(* IEC 61131-3 sources: TIA2AX/tests/V18/test_projects/expected/HW_2200330/ST40_PLC, 7 files *)

(* ---- HwIdentifiers.st ---- *)
TYPE
	HwIdentifiers : WORD
	(
		ST40_PLC_Profilschiene_0 :=	WORD#256,
		ST40_PLC :=	WORD#48,
		ST40_PLC_Card_reader_writer_1 :=	WORD#51,
		ST40_PLC_CPU_display_1 :=	WORD#54,
		ST40_PLC_OPC_UA_1 :=	WORD#117,
		ST40_PLC_DP_interface_1 :=	WORD#60,
		ST40_PLC_PROFINET_interface_1 :=	WORD#64,
		ST40_PLC_PROFINET_interface_1_Port_1 :=	WORD#65,
		ST40_PLC_PROFINET_interface_1_Port_2 :=	WORD#66,
		ST40_PLC_PROFINET_interface_2 :=	WORD#72,
		ST40_PLC_PROFINET_interface_2_Port_1 :=	WORD#73,
		ST40_Switch_SCALANCE_X_rack :=	WORD#415,
		ST40_Switch :=	WORD#416,
		ST40_Switch_ST40_Switch :=	WORD#417,
		ST40_Switch_SCALANCE_interface_1 :=	WORD#418,
		ST40_Switch_SCALANCE_interface_1_Port_1 :=	WORD#419,
		ST40_Switch_SCALANCE_interface_1_Port_2 :=	WORD#420,
		ST40_Switch_SCALANCE_interface_1_Port_3 :=	WORD#421,
		ST40_Switch_SCALANCE_interface_1_Port_4 :=	WORD#422,
		ST40_Switch_SCALANCE_interface_1_Port_5 :=	WORD#423,
		ST40_Switch_SCALANCE_interface_1_Port_6 :=	WORD#424,
		ST40_Switch_SCALANCE_interface_1_Port_7 :=	WORD#425,
		ST40_Switch_SCALANCE_interface_1_Port_8 :=	WORD#426,
		ST40_Switch_SCALANCE_interface_1_Port_9 :=	WORD#427,
		ST40_Switch_SCALANCE_interface_1_Port_10 :=	WORD#428,
		ST40_Switch_SCALANCE_interface_1_Port_11 :=	WORD#429,
		ST40_Switch_SCALANCE_interface_1_Port_12 :=	WORD#430,
		ST40_Switch_SCALANCE_interface_1_Port_13 :=	WORD#431,
		ST40_Switch_SCALANCE_interface_1_Port_14 :=	WORD#432,
		ST40_Switch_SCALANCE_interface_1_Port_15 :=	WORD#433,
		ST40_Switch_SCALANCE_interface_1_Port_16 :=	WORD#434,
		ST40_2_DM260_Rack :=	WORD#270,
		ST40_2_DM260 :=	WORD#258,
		ST40_2_DM260_Interface :=	WORD#259,
		ST40_2_DM260_Interface_Port_1 :=	WORD#260,
		ST40_2_DM260_DataMan_260 :=	WORD#261,
		ST40_2_DM260_Acquisition_Control_1 :=	WORD#262,
		ST40_2_DM260_Acquisition_Status_1 :=	WORD#263,
		ST40_2_DM260_Results_Control_1 :=	WORD#264,
		ST40_2_DM260_Results_Status_1 :=	WORD#265,
		ST40_2_DM260_Soft_Event_Control_1 :=	WORD#266,
		ST40_2_DM260_User_Data_64_bytes_1 :=	WORD#267,
		ST40_2_DM260_Result_Data_64_bytes_1 :=	WORD#268,
		ST40_3_DM260_Rack :=	WORD#272,
		ST40_3_DM260 :=	WORD#273,
		ST40_3_DM260_Interface :=	WORD#274,
		ST40_3_DM260_Interface_Port_1 :=	WORD#275,
		ST40_3_DM260_DataMan_260 :=	WORD#276,
		ST40_3_DM260_Acquisition_Control_1 :=	WORD#277,
		ST40_3_DM260_Acquisition_Status_1 :=	WORD#278,
		ST40_3_DM260_Results_Control_1 :=	WORD#279,
		ST40_3_DM260_Results_Status_1 :=	WORD#280,
		ST40_3_DM260_Soft_Event_Control_1 :=	WORD#281,
		ST40_3_DM260_User_Data_64_bytes_1 :=	WORD#282,
		ST40_3_DM260_Result_Data_64_bytes_1 :=	WORD#283,
		ST40_1_DM260_Rack :=	WORD#285,
		ST40_1_DM260 :=	WORD#286,
		ST40_1_DM260_Interface :=	WORD#287,
		ST40_1_DM260_Interface_Port_1 :=	WORD#288,
		ST40_1_DM260_DataMan_260 :=	WORD#289,
		ST40_1_DM260_Acquisition_Control_1 :=	WORD#290,
		ST40_1_DM260_Acquisition_Status_1 :=	WORD#291,
		ST40_1_DM260_Results_Control_1 :=	WORD#292,
		ST40_1_DM260_Results_Status_1 :=	WORD#293,
		ST40_1_DM260_Soft_Event_Control_1 :=	WORD#294,
		ST40_1_DM260_User_Data_64_bytes_1 :=	WORD#295,
		ST40_1_DM260_Result_Data_64_bytes_1 :=	WORD#296,
		ST40_2_CMMT_2GF2_Promess_PN_IO_Interface :=	WORD#300,
		ST40_2_CMMT_2GF2_Promess_PN_IO_Interface_Port_1 :=	WORD#301,
		ST40_2_CMMT_2GF2_Promess_PN_IO_Interface_Port_2 :=	WORD#302,
		ST40_2_CMMT_2GF2_Promess_CMMT_AS_V1 :=	WORD#303,
		ST40_2_CMMT_2GF2_Promess_DO_SERVO_1_Module_Access_Point :=	WORD#305,
		ST40_2_CMMT_2GF2_Promess_DO_SERVO_1_Siemens_telegram_111_PZD_12_12 :=	WORD#306,
		ST40_2_CMMT_2GF2_Promess_Siemens_telegram_111_PZD_12_12 :=	WORD#306,
		ST40_2_Promess_Rack :=	WORD#328,
		ST40_2_Promess :=	WORD#329,
		ST40_2_Promess_X1 :=	WORD#330,
		ST40_2_Promess_X1_X1_P1 :=	WORD#331,
		ST40_2_Promess_X1_X1_P2 :=	WORD#332,
		ST40_2_Promess_UniDrive_M :=	WORD#333,
		ST40_2_Promess_Menu_30_01_In_1 :=	WORD#334,
		ST40_2_Promess_Menu_30_02_In_1 :=	WORD#335,
		ST40_2_Promess_Menu_30_03_In_1 :=	WORD#336,
		ST40_2_Promess_Menu_30_04_In_1 :=	WORD#337,
		ST40_2_Promess_Menu_30_05_In_1 :=	WORD#338,
		ST40_2_Promess_Menu_30_06_In_1 :=	WORD#339,
		ST40_2_Promess_Menu_30_07_In_1 :=	WORD#340,
		ST40_2_Promess_Menu_30_08_In_1 :=	WORD#341,
		ST40_2_Promess_Menu_30_09_In_1 :=	WORD#342,
		ST40_2_Promess_Menu_30_10_In_1 :=	WORD#343,
		ST40_2_Promess_Menu_30_11_In_1 :=	WORD#344,
		ST40_2_Promess_Menu_30_12_In_1 :=	WORD#345,
		ST40_2_Promess_Menu_30_13_In_1 :=	WORD#346,
		ST40_2_Promess_Menu_30_14_In_1 :=	WORD#347,
		ST40_2_Promess_Menu_30_15_In_1 :=	WORD#348,
		ST40_2_Promess_Menu_30_16_In_1 :=	WORD#349,
		ST40_2_Promess_Menu_30_33_Out_1 :=	WORD#350,
		ST40_2_Promess_Menu_30_34_Out_1 :=	WORD#351,
		ST40_2_Promess_Menu_30_35_Out_1 :=	WORD#352,
		ST40_2_Promess_Menu_30_36_Out_1 :=	WORD#353,
		ST40_2_Promess_Menu_30_37_Out_1 :=	WORD#354,
		ST40_2_Promess_Menu_30_38_Out_1 :=	WORD#355,
		ST40_2_Promess_Menu_30_39_Out_1 :=	WORD#356,
		ST40_2_Promess_Menu_30_40_Out_1 :=	WORD#357,
		ST40_2_Promess_Menu_30_41_Out_1 :=	WORD#358,
		ST40_2_Promess_Menu_30_42_Out_1 :=	WORD#359,
		ST40_2_Promess_Menu_30_43_Out_1 :=	WORD#360,
		ST40_2_Promess_Menu_30_44_Out_1 :=	WORD#361,
		ST40_2_Promess_Menu_30_45_Out_1 :=	WORD#362,
		ST40_2_Promess_Menu_30_46_Out_1 :=	WORD#363,
		ST40_2_Promess_Menu_30_47_Out_1 :=	WORD#364,
		ST40_2_Promess_Menu_30_48_Out_1 :=	WORD#365,
		ST40_2_Promess_Menu_30_17_In_1 :=	WORD#366,
		ST40_2_Promess_Menu_30_18_In_1 :=	WORD#367,
		ST40_2_Promess_Menu_30_19_In_1 :=	WORD#368,
		ST40_2_Promess_Menu_30_20_In_1 :=	WORD#369,
		ST40_2_Promess_Menu_30_21_In_1 :=	WORD#370,
		ST40_2_Promess_Menu_30_22_In_1 :=	WORD#371,
		ST40_2_Promess_Menu_30_23_In_1 :=	WORD#372,
		ST40_2_Promess_Menu_30_24_In_1 :=	WORD#373,
		ST40_2_Promess_Menu_30_25_In_1 :=	WORD#374,
		ST40_2_Promess_Menu_30_26_In_1 :=	WORD#375,
		ST40_2_Promess_Menu_30_27_In_1 :=	WORD#376,
		ST40_2_Promess_Menu_30_28_In_1 :=	WORD#377,
		ST40_2_Promess_Menu_30_29_In_1 :=	WORD#307,
		ST40_2_Promess_Menu_30_30_In_1 :=	WORD#308,
		ST40_2_Promess_Menu_30_31_In_1 :=	WORD#309,
		ST40_2_Promess_Menu_30_32_In_1 :=	WORD#310,
		ST40_2_Promess_Menu_30_49_Out_1 :=	WORD#311,
		ST40_2_Promess_Menu_30_50_Out_1 :=	WORD#312,
		ST40_2_Promess_Menu_30_51_Out_1 :=	WORD#313,
		ST40_2_Promess_Menu_30_52_Out_1 :=	WORD#314,
		ST40_2_Promess_Menu_30_53_Out_1 :=	WORD#315,
		ST40_2_Promess_Menu_30_54_Out_1 :=	WORD#316,
		ST40_2_Promess_Menu_30_55_Out_1 :=	WORD#317,
		ST40_2_Promess_Menu_30_56_Out_1 :=	WORD#318,
		ST40_2_Promess_Menu_30_57_Out_1 :=	WORD#319,
		ST40_2_Promess_Menu_30_58_Out_1 :=	WORD#320,
		ST40_2_Promess_Menu_30_59_Out_1 :=	WORD#321,
		ST40_2_Promess_Menu_30_60_Out_1 :=	WORD#322,
		ST40_2_Promess_Menu_30_61_Out_1 :=	WORD#323,
		ST40_2_Promess_Menu_30_62_Out_1 :=	WORD#324,
		ST40_2_Promess_Menu_30_63_Out_1 :=	WORD#325,
		ST40_2_Promess_Menu_30_64_Out_1 :=	WORD#326,
		ST40_CPX_PN_IO_Interface :=	WORD#381,
		ST40_CPX_PN_IO_Interface_Port_1 :=	WORD#382,
		ST40_CPX_PN_IO_Interface_Port_2 :=	WORD#383,
		ST40_CPX_CPX :=	WORD#384,
		ST40_CPX_MPA1S_VMPA1_FB_EMS_8_8DO_1 :=	WORD#385,
		ST40_CPX_MPA1S_VMPA1_FB_EMS_8_8DO_2 :=	WORD#386,
		ST40_CPX_MPA1S_VMPA1_FB_EMS_8_8DO_3 :=	WORD#387,
		ST40_CPX_MPA1G_VMPA1_FB_EMG_8_8DO_1 :=	WORD#388,
		ST40_ET200SP_Rack_0 :=	WORD#390,
		ST40_ET200SP :=	WORD#391,
		ST40_ET200SP_ST40_ET200SP :=	WORD#392,
		ST40_ET200SP_PROFINET_interface :=	WORD#393,
		ST40_ET200SP_PROFINET_interface_Port_1 :=	WORD#395,
		ST40_ET200SP_PROFINET_interface_Port_2 :=	WORD#394,
		ST40_ET200SP_BA_2xRJ45 :=	WORD#395,
		ST40_ET200SP_CM_4xIO_Link_1 :=	WORD#396,
		ST40_ET200SP_CM_4xIO_Link_2 :=	WORD#397,
		ST40_ET200SP_DI_8x24VDC_ST_1 :=	WORD#398,
		ST40_ET200SP_DI_8x24VDC_ST_2 :=	WORD#399,
		ST40_ET200SP_DI_16x24VDC_ST_1 :=	WORD#400,
		ST40_ET200SP_DI_8x24VDC_ST_3 :=	WORD#401,
		ST40_ET200SP_DQ_16x24VDC_0_5A_ST_1 :=	WORD#402,
		ST40_ET200SP_DQ_8x24VDC_0_5A_ST_2 :=	WORD#403,
		ST40_ET200SP_DQ_8x24VDC_0_5A_ST_3 :=	WORD#404,
		ST40_ET200SP_Servermodul_1 :=	WORD#405,
		ST40_HMI_ConnectionBox_Connection_Box :=	WORD#407,
		ST40_HMI_ConnectionBox :=	WORD#408,
		ST40_HMI_ConnectionBox_ST40_HMI_ConnectionBox :=	WORD#409,
		ST40_HMI_ConnectionBox_SCALANCE_interface_1 :=	WORD#410,
		ST40_HMI_ConnectionBox_SCALANCE_interface_1_Port_1 :=	WORD#411,
		ST40_HMI_ConnectionBox_SCALANCE_interface_1_Port_2 :=	WORD#412,
		ST40_HMI_ConnectionBox_SCALANCE_interface_1_Port_3 :=	WORD#413,
		NONE:= WORD#0
	);
END_TYPE

(* ---- HwInputs.st ---- *)
TYPE
	HwInputs : STRUCT
		ST40_2_DM260_Acquisition_Status_1 AT %B2500 : ARRAY[0..2] OF BYTE;
		ST40_2_DM260_Results_Status_1 AT %B2503 : BYTE;
		ST40_2_DM260_Soft_Event_Control_1 AT %B2504 : BYTE;
		ST40_2_DM260_Result_Data_64_bytes_1 AT %B2510 : ARRAY[0..71] OF BYTE;
		ST40_3_DM260_Acquisition_Status_1 AT %B3500 : ARRAY[0..2] OF BYTE;
		ST40_3_DM260_Results_Status_1 AT %B3503 : BYTE;
		ST40_3_DM260_Soft_Event_Control_1 AT %B3504 : BYTE;
		ST40_3_DM260_Result_Data_64_bytes_1 AT %B3510 : ARRAY[0..71] OF BYTE;
		ST40_1_DM260_Acquisition_Status_1 AT %B1600 : ARRAY[0..2] OF BYTE;
		ST40_1_DM260_Results_Status_1 AT %B1603 : BYTE;
		ST40_1_DM260_Soft_Event_Control_1 AT %B1604 : BYTE;
		ST40_1_DM260_Result_Data_64_bytes_1 AT %B1610 : ARRAY[0..71] OF BYTE;
		ST40_2_CMMT_2GF2_Promess_DO_SERVO_1_Siemens_telegram_111_PZD_12_12 AT %B1100 : ARRAY[0..23] OF BYTE;
		ST40_2_Promess_Menu_30_01_In_1 AT %B2100 : WORD;
		ST40_2_Promess_Menu_30_02_In_1 AT %B2102 : WORD;
		ST40_2_Promess_Menu_30_03_In_1 AT %B2104 : WORD;
		ST40_2_Promess_Menu_30_04_In_1 AT %B2106 : WORD;
		ST40_2_Promess_Menu_30_05_In_1 AT %B2108 : WORD;
		ST40_2_Promess_Menu_30_06_In_1 AT %B2110 : WORD;
		ST40_2_Promess_Menu_30_07_In_1 AT %B2112 : WORD;
		ST40_2_Promess_Menu_30_08_In_1 AT %B2114 : WORD;
		ST40_2_Promess_Menu_30_09_In_1 AT %B2116 : WORD;
		ST40_2_Promess_Menu_30_10_In_1 AT %B2118 : WORD;
		ST40_2_Promess_Menu_30_11_In_1 AT %B2120 : WORD;
		ST40_2_Promess_Menu_30_12_In_1 AT %B2122 : WORD;
		ST40_2_Promess_Menu_30_13_In_1 AT %B2124 : WORD;
		ST40_2_Promess_Menu_30_14_In_1 AT %B2126 : WORD;
		ST40_2_Promess_Menu_30_15_In_1 AT %B2128 : WORD;
		ST40_2_Promess_Menu_30_16_In_1 AT %B2130 : WORD;
		ST40_2_Promess_Menu_30_17_In_1 AT %B2132 : WORD;
		ST40_2_Promess_Menu_30_18_In_1 AT %B2134 : WORD;
		ST40_2_Promess_Menu_30_19_In_1 AT %B2136 : WORD;
		ST40_2_Promess_Menu_30_20_In_1 AT %B2138 : WORD;
		ST40_2_Promess_Menu_30_21_In_1 AT %B2140 : WORD;
		ST40_2_Promess_Menu_30_22_In_1 AT %B2142 : WORD;
		ST40_2_Promess_Menu_30_23_In_1 AT %B2144 : WORD;
		ST40_2_Promess_Menu_30_24_In_1 AT %B2146 : WORD;
		ST40_2_Promess_Menu_30_25_In_1 AT %B2148 : WORD;
		ST40_2_Promess_Menu_30_26_In_1 AT %B2150 : WORD;
		ST40_2_Promess_Menu_30_27_In_1 AT %B2152 : WORD;
		ST40_2_Promess_Menu_30_28_In_1 AT %B2154 : WORD;
		ST40_2_Promess_Menu_30_29_In_1 AT %B2156 : WORD;
		ST40_2_Promess_Menu_30_30_In_1 AT %B2158 : WORD;
		ST40_2_Promess_Menu_30_31_In_1 AT %B2160 : WORD;
		ST40_2_Promess_Menu_30_32_In_1 AT %B2162 : WORD;
		ST40_ET200SP_CM_4xIO_Link_1 AT %B100 : ARRAY[0..31] OF BYTE;
		ST40_ET200SP_CM_4xIO_Link_2 AT %B132 : ARRAY[0..31] OF BYTE;
		ST40_ET200SP_DI_8x24VDC_ST_1 AT %B0 : BYTE;
		ST40_ET200SP_DI_8x24VDC_ST_2 AT %B1 : BYTE;
		ST40_ET200SP_DI_16x24VDC_ST_1 AT %B2 : WORD;
		ST40_ET200SP_DI_8x24VDC_ST_3 AT %B4 : BYTE;
	END_STRUCT;
END_TYPE

(* ---- HwOutputs.st ---- *)
TYPE
	HwOutputs : STRUCT
		ST40_2_DM260_Acquisition_Control_1 AT %B2500 : BYTE;
		ST40_2_DM260_Results_Control_1 AT %B2503 : BYTE;
		ST40_2_DM260_Soft_Event_Control_1 AT %B2504 : BYTE;
		ST40_2_DM260_User_Data_64_bytes_1 AT %B2510 : ARRAY[0..67] OF BYTE;
		ST40_3_DM260_Acquisition_Control_1 AT %B3500 : BYTE;
		ST40_3_DM260_Results_Control_1 AT %B3503 : BYTE;
		ST40_3_DM260_Soft_Event_Control_1 AT %B3504 : BYTE;
		ST40_3_DM260_User_Data_64_bytes_1 AT %B3510 : ARRAY[0..67] OF BYTE;
		ST40_1_DM260_Acquisition_Control_1 AT %B1600 : BYTE;
		ST40_1_DM260_Results_Control_1 AT %B1603 : BYTE;
		ST40_1_DM260_Soft_Event_Control_1 AT %B1604 : BYTE;
		ST40_1_DM260_User_Data_64_bytes_1 AT %B1610 : ARRAY[0..67] OF BYTE;
		ST40_2_CMMT_2GF2_Promess_DO_SERVO_1_Siemens_telegram_111_PZD_12_12 AT %B1100 : ARRAY[0..23] OF BYTE;
		ST40_2_Promess_Menu_30_33_Out_1 AT %B2100 : WORD;
		ST40_2_Promess_Menu_30_34_Out_1 AT %B2102 : WORD;
		ST40_2_Promess_Menu_30_35_Out_1 AT %B2104 : WORD;
		ST40_2_Promess_Menu_30_36_Out_1 AT %B2106 : WORD;
		ST40_2_Promess_Menu_30_37_Out_1 AT %B2108 : WORD;
		ST40_2_Promess_Menu_30_38_Out_1 AT %B2110 : WORD;
		ST40_2_Promess_Menu_30_39_Out_1 AT %B2112 : WORD;
		ST40_2_Promess_Menu_30_40_Out_1 AT %B2114 : WORD;
		ST40_2_Promess_Menu_30_41_Out_1 AT %B2116 : WORD;
		ST40_2_Promess_Menu_30_42_Out_1 AT %B2118 : WORD;
		ST40_2_Promess_Menu_30_43_Out_1 AT %B2120 : WORD;
		ST40_2_Promess_Menu_30_44_Out_1 AT %B2122 : WORD;
		ST40_2_Promess_Menu_30_45_Out_1 AT %B2124 : WORD;
		ST40_2_Promess_Menu_30_46_Out_1 AT %B2126 : WORD;
		ST40_2_Promess_Menu_30_47_Out_1 AT %B2128 : WORD;
		ST40_2_Promess_Menu_30_48_Out_1 AT %B2130 : WORD;
		ST40_2_Promess_Menu_30_49_Out_1 AT %B2132 : WORD;
		ST40_2_Promess_Menu_30_50_Out_1 AT %B2134 : WORD;
		ST40_2_Promess_Menu_30_51_Out_1 AT %B2136 : WORD;
		ST40_2_Promess_Menu_30_52_Out_1 AT %B2138 : WORD;
		ST40_2_Promess_Menu_30_53_Out_1 AT %B2140 : WORD;
		ST40_2_Promess_Menu_30_54_Out_1 AT %B2142 : WORD;
		ST40_2_Promess_Menu_30_55_Out_1 AT %B2144 : WORD;
		ST40_2_Promess_Menu_30_56_Out_1 AT %B2146 : WORD;
		ST40_2_Promess_Menu_30_57_Out_1 AT %B2148 : WORD;
		ST40_2_Promess_Menu_30_58_Out_1 AT %B2150 : WORD;
		ST40_2_Promess_Menu_30_59_Out_1 AT %B2152 : WORD;
		ST40_2_Promess_Menu_30_60_Out_1 AT %B2154 : WORD;
		ST40_2_Promess_Menu_30_61_Out_1 AT %B2156 : WORD;
		ST40_2_Promess_Menu_30_62_Out_1 AT %B2158 : WORD;
		ST40_2_Promess_Menu_30_63_Out_1 AT %B2160 : WORD;
		ST40_2_Promess_Menu_30_64_Out_1 AT %B2162 : WORD;
		ST40_CPX_MPA1S_VMPA1_FB_EMS_8_8DO_1 AT %B200 : BYTE;
		ST40_CPX_MPA1S_VMPA1_FB_EMS_8_8DO_2 AT %B201 : BYTE;
		ST40_CPX_MPA1S_VMPA1_FB_EMS_8_8DO_3 AT %B202 : BYTE;
		ST40_CPX_MPA1G_VMPA1_FB_EMG_8_8DO_1 AT %B203 : BYTE;
		ST40_ET200SP_CM_4xIO_Link_1 AT %B100 : ARRAY[0..31] OF BYTE;
		ST40_ET200SP_CM_4xIO_Link_2 AT %B132 : ARRAY[0..31] OF BYTE;
		ST40_ET200SP_DQ_16x24VDC_0_5A_ST_1 AT %B0 : WORD;
		ST40_ET200SP_DQ_8x24VDC_0_5A_ST_2 AT %B2 : BYTE;
		ST40_ET200SP_DQ_8x24VDC_0_5A_ST_3 AT %B3 : BYTE;
	END_STRUCT;
END_TYPE

(* ---- PlcInputs.st ---- *)
TYPE
	PlcInputs : STRUCT
		ST40_2_DM260_Acquisition_Status_1 : ARRAY[0..2] OF BYTE;
		ST40_2_DM260_Results_Status_1 : BYTE;
		ST40_2_DM260_Soft_Event_Control_1 : BYTE;
		ST40_2_DM260_Result_Data_64_bytes_1 : ARRAY[0..71] OF BYTE;
		ST40_3_DM260_Acquisition_Status_1 : ARRAY[0..2] OF BYTE;
		ST40_3_DM260_Results_Status_1 : BYTE;
		ST40_3_DM260_Soft_Event_Control_1 : BYTE;
		ST40_3_DM260_Result_Data_64_bytes_1 : ARRAY[0..71] OF BYTE;
		ST40_1_DM260_Acquisition_Status_1 : ARRAY[0..2] OF BYTE;
		ST40_1_DM260_Results_Status_1 : BYTE;
		ST40_1_DM260_Soft_Event_Control_1 : BYTE;
		ST40_1_DM260_Result_Data_64_bytes_1 : ARRAY[0..71] OF BYTE;
		ST40_2_CMMT_2GF2_Promess_DO_SERVO_1_Siemens_telegram_111_PZD_12_12 : ARRAY[0..23] OF BYTE;
		ST40_2_Promess_Menu_30_01_In_1 : WORD;
		ST40_2_Promess_Menu_30_02_In_1 : WORD;
		ST40_2_Promess_Menu_30_03_In_1 : WORD;
		ST40_2_Promess_Menu_30_04_In_1 : WORD;
		ST40_2_Promess_Menu_30_05_In_1 : WORD;
		ST40_2_Promess_Menu_30_06_In_1 : WORD;
		ST40_2_Promess_Menu_30_07_In_1 : WORD;
		ST40_2_Promess_Menu_30_08_In_1 : WORD;
		ST40_2_Promess_Menu_30_09_In_1 : WORD;
		ST40_2_Promess_Menu_30_10_In_1 : WORD;
		ST40_2_Promess_Menu_30_11_In_1 : WORD;
		ST40_2_Promess_Menu_30_12_In_1 : WORD;
		ST40_2_Promess_Menu_30_13_In_1 : WORD;
		ST40_2_Promess_Menu_30_14_In_1 : WORD;
		ST40_2_Promess_Menu_30_15_In_1 : WORD;
		ST40_2_Promess_Menu_30_16_In_1 : WORD;
		ST40_2_Promess_Menu_30_17_In_1 : WORD;
		ST40_2_Promess_Menu_30_18_In_1 : WORD;
		ST40_2_Promess_Menu_30_19_In_1 : WORD;
		ST40_2_Promess_Menu_30_20_In_1 : WORD;
		ST40_2_Promess_Menu_30_21_In_1 : WORD;
		ST40_2_Promess_Menu_30_22_In_1 : WORD;
		ST40_2_Promess_Menu_30_23_In_1 : WORD;
		ST40_2_Promess_Menu_30_24_In_1 : WORD;
		ST40_2_Promess_Menu_30_25_In_1 : WORD;
		ST40_2_Promess_Menu_30_26_In_1 : WORD;
		ST40_2_Promess_Menu_30_27_In_1 : WORD;
		ST40_2_Promess_Menu_30_28_In_1 : WORD;
		ST40_2_Promess_Menu_30_29_In_1 : WORD;
		ST40_2_Promess_Menu_30_30_In_1 : WORD;
		ST40_2_Promess_Menu_30_31_In_1 : WORD;
		ST40_2_Promess_Menu_30_32_In_1 : WORD;
		ST40_ET200SP_CM_4xIO_Link_1 : ARRAY[0..31] OF BYTE;
		ST40_ET200SP_CM_4xIO_Link_2 : ARRAY[0..31] OF BYTE;
		ST40_ET200SP_DI_8x24VDC_ST_1 : BYTE;
		ST40_ET200SP_DI_8x24VDC_ST_2 : BYTE;
		ST40_ET200SP_DI_16x24VDC_ST_1 : WORD;
		ST40_ET200SP_DI_8x24VDC_ST_3 : BYTE;
	END_STRUCT;
END_TYPE

(* ---- PlcOutputs.st ---- *)
TYPE
	PlcOutputs : STRUCT
		ST40_2_DM260_Acquisition_Control_1 : BYTE;
		ST40_2_DM260_Results_Control_1 : BYTE;
		ST40_2_DM260_Soft_Event_Control_1 : BYTE;
		ST40_2_DM260_User_Data_64_bytes_1 : ARRAY[0..67] OF BYTE;
		ST40_3_DM260_Acquisition_Control_1 : BYTE;
		ST40_3_DM260_Results_Control_1 : BYTE;
		ST40_3_DM260_Soft_Event_Control_1 : BYTE;
		ST40_3_DM260_User_Data_64_bytes_1 : ARRAY[0..67] OF BYTE;
		ST40_1_DM260_Acquisition_Control_1 : BYTE;
		ST40_1_DM260_Results_Control_1 : BYTE;
		ST40_1_DM260_Soft_Event_Control_1 : BYTE;
		ST40_1_DM260_User_Data_64_bytes_1 : ARRAY[0..67] OF BYTE;
		ST40_2_CMMT_2GF2_Promess_DO_SERVO_1_Siemens_telegram_111_PZD_12_12 : ARRAY[0..23] OF BYTE;
		ST40_2_Promess_Menu_30_33_Out_1 : WORD;
		ST40_2_Promess_Menu_30_34_Out_1 : WORD;
		ST40_2_Promess_Menu_30_35_Out_1 : WORD;
		ST40_2_Promess_Menu_30_36_Out_1 : WORD;
		ST40_2_Promess_Menu_30_37_Out_1 : WORD;
		ST40_2_Promess_Menu_30_38_Out_1 : WORD;
		ST40_2_Promess_Menu_30_39_Out_1 : WORD;
		ST40_2_Promess_Menu_30_40_Out_1 : WORD;
		ST40_2_Promess_Menu_30_41_Out_1 : WORD;
		ST40_2_Promess_Menu_30_42_Out_1 : WORD;
		ST40_2_Promess_Menu_30_43_Out_1 : WORD;
		ST40_2_Promess_Menu_30_44_Out_1 : WORD;
		ST40_2_Promess_Menu_30_45_Out_1 : WORD;
		ST40_2_Promess_Menu_30_46_Out_1 : WORD;
		ST40_2_Promess_Menu_30_47_Out_1 : WORD;
		ST40_2_Promess_Menu_30_48_Out_1 : WORD;
		ST40_2_Promess_Menu_30_49_Out_1 : WORD;
		ST40_2_Promess_Menu_30_50_Out_1 : WORD;
		ST40_2_Promess_Menu_30_51_Out_1 : WORD;
		ST40_2_Promess_Menu_30_52_Out_1 : WORD;
		ST40_2_Promess_Menu_30_53_Out_1 : WORD;
		ST40_2_Promess_Menu_30_54_Out_1 : WORD;
		ST40_2_Promess_Menu_30_55_Out_1 : WORD;
		ST40_2_Promess_Menu_30_56_Out_1 : WORD;
		ST40_2_Promess_Menu_30_57_Out_1 : WORD;
		ST40_2_Promess_Menu_30_58_Out_1 : WORD;
		ST40_2_Promess_Menu_30_59_Out_1 : WORD;
		ST40_2_Promess_Menu_30_60_Out_1 : WORD;
		ST40_2_Promess_Menu_30_61_Out_1 : WORD;
		ST40_2_Promess_Menu_30_62_Out_1 : WORD;
		ST40_2_Promess_Menu_30_63_Out_1 : WORD;
		ST40_2_Promess_Menu_30_64_Out_1 : WORD;
		ST40_CPX_MPA1S_VMPA1_FB_EMS_8_8DO_1 : BYTE;
		ST40_CPX_MPA1S_VMPA1_FB_EMS_8_8DO_2 : BYTE;
		ST40_CPX_MPA1S_VMPA1_FB_EMS_8_8DO_3 : BYTE;
		ST40_CPX_MPA1G_VMPA1_FB_EMG_8_8DO_1 : BYTE;
		ST40_ET200SP_CM_4xIO_Link_1 : ARRAY[0..31] OF BYTE;
		ST40_ET200SP_CM_4xIO_Link_2 : ARRAY[0..31] OF BYTE;
		ST40_ET200SP_DQ_16x24VDC_0_5A_ST_1 : WORD;
		ST40_ET200SP_DQ_8x24VDC_0_5A_ST_2 : BYTE;
		ST40_ET200SP_DQ_8x24VDC_0_5A_ST_3 : BYTE;
	END_STRUCT;
END_TYPE

(* ---- CopyInputs.st ---- *)
FUNCTION CopyInputs
	VAR_EXTERNAL
		HwInputs : HwInputs;
		PlcInputs : PlcInputs;
	END_VAR
	PlcInputs.ST40_2_DM260_Acquisition_Status_1[0] := HwInputs.ST40_2_DM260_Acquisition_Status_1[0];
	PlcInputs.ST40_2_DM260_Acquisition_Status_1[1] := HwInputs.ST40_2_DM260_Acquisition_Status_1[1];
	PlcInputs.ST40_2_DM260_Acquisition_Status_1[2] := HwInputs.ST40_2_DM260_Acquisition_Status_1[2];
	PlcInputs.ST40_2_DM260_Results_Status_1 := HwInputs.ST40_2_DM260_Results_Status_1;
	PlcInputs.ST40_2_DM260_Soft_Event_Control_1 := HwInputs.ST40_2_DM260_Soft_Event_Control_1;
	PlcInputs.ST40_2_DM260_Result_Data_64_bytes_1[0] := HwInputs.ST40_2_DM260_Result_Data_64_bytes_1[0];
	PlcInputs.ST40_2_DM260_Result_Data_64_bytes_1[1] := HwInputs.ST40_2_DM260_Result_Data_64_bytes_1[1];
	PlcInputs.ST40_2_DM260_Result_Data_64_bytes_1[2] := HwInputs.ST40_2_DM260_Result_Data_64_bytes_1[2];
	PlcInputs.ST40_2_DM260_Result_Data_64_bytes_1[3] := HwInputs.ST40_2_DM260_Result_Data_64_bytes_1[3];
	PlcInputs.ST40_2_DM260_Result_Data_64_bytes_1[4] := HwInputs.ST40_2_DM260_Result_Data_64_bytes_1[4];
	PlcInputs.ST40_2_DM260_Result_Data_64_bytes_1[5] := HwInputs.ST40_2_DM260_Result_Data_64_bytes_1[5];
	PlcInputs.ST40_2_DM260_Result_Data_64_bytes_1[6] := HwInputs.ST40_2_DM260_Result_Data_64_bytes_1[6];
	PlcInputs.ST40_2_DM260_Result_Data_64_bytes_1[7] := HwInputs.ST40_2_DM260_Result_Data_64_bytes_1[7];
	PlcInputs.ST40_2_DM260_Result_Data_64_bytes_1[8] := HwInputs.ST40_2_DM260_Result_Data_64_bytes_1[8];
	PlcInputs.ST40_2_DM260_Result_Data_64_bytes_1[9] := HwInputs.ST40_2_DM260_Result_Data_64_bytes_1[9];
	PlcInputs.ST40_2_DM260_Result_Data_64_bytes_1[10] := HwInputs.ST40_2_DM260_Result_Data_64_bytes_1[10];
	PlcInputs.ST40_2_DM260_Result_Data_64_bytes_1[11] := HwInputs.ST40_2_DM260_Result_Data_64_bytes_1[11];
	PlcInputs.ST40_2_DM260_Result_Data_64_bytes_1[12] := HwInputs.ST40_2_DM260_Result_Data_64_bytes_1[12];
	PlcInputs.ST40_2_DM260_Result_Data_64_bytes_1[13] := HwInputs.ST40_2_DM260_Result_Data_64_bytes_1[13];
	PlcInputs.ST40_2_DM260_Result_Data_64_bytes_1[14] := HwInputs.ST40_2_DM260_Result_Data_64_bytes_1[14];
	PlcInputs.ST40_2_DM260_Result_Data_64_bytes_1[15] := HwInputs.ST40_2_DM260_Result_Data_64_bytes_1[15];
	PlcInputs.ST40_2_DM260_Result_Data_64_bytes_1[16] := HwInputs.ST40_2_DM260_Result_Data_64_bytes_1[16];
	PlcInputs.ST40_2_DM260_Result_Data_64_bytes_1[17] := HwInputs.ST40_2_DM260_Result_Data_64_bytes_1[17];
	PlcInputs.ST40_2_DM260_Result_Data_64_bytes_1[18] := HwInputs.ST40_2_DM260_Result_Data_64_bytes_1[18];
	PlcInputs.ST40_2_DM260_Result_Data_64_bytes_1[19] := HwInputs.ST40_2_DM260_Result_Data_64_bytes_1[19];
	PlcInputs.ST40_2_DM260_Result_Data_64_bytes_1[20] := HwInputs.ST40_2_DM260_Result_Data_64_bytes_1[20];
	PlcInputs.ST40_2_DM260_Result_Data_64_bytes_1[21] := HwInputs.ST40_2_DM260_Result_Data_64_bytes_1[21];
	PlcInputs.ST40_2_DM260_Result_Data_64_bytes_1[22] := HwInputs.ST40_2_DM260_Result_Data_64_bytes_1[22];
	PlcInputs.ST40_2_DM260_Result_Data_64_bytes_1[23] := HwInputs.ST40_2_DM260_Result_Data_64_bytes_1[23];
	PlcInputs.ST40_2_DM260_Result_Data_64_bytes_1[24] := HwInputs.ST40_2_DM260_Result_Data_64_bytes_1[24];
	PlcInputs.ST40_2_DM260_Result_Data_64_bytes_1[25] := HwInputs.ST40_2_DM260_Result_Data_64_bytes_1[25];
	PlcInputs.ST40_2_DM260_Result_Data_64_bytes_1[26] := HwInputs.ST40_2_DM260_Result_Data_64_bytes_1[26];
	PlcInputs.ST40_2_DM260_Result_Data_64_bytes_1[27] := HwInputs.ST40_2_DM260_Result_Data_64_bytes_1[27];
	PlcInputs.ST40_2_DM260_Result_Data_64_bytes_1[28] := HwInputs.ST40_2_DM260_Result_Data_64_bytes_1[28];
	PlcInputs.ST40_2_DM260_Result_Data_64_bytes_1[29] := HwInputs.ST40_2_DM260_Result_Data_64_bytes_1[29];
	PlcInputs.ST40_2_DM260_Result_Data_64_bytes_1[30] := HwInputs.ST40_2_DM260_Result_Data_64_bytes_1[30];
	PlcInputs.ST40_2_DM260_Result_Data_64_bytes_1[31] := HwInputs.ST40_2_DM260_Result_Data_64_bytes_1[31];
	PlcInputs.ST40_2_DM260_Result_Data_64_bytes_1[32] := HwInputs.ST40_2_DM260_Result_Data_64_bytes_1[32];
	PlcInputs.ST40_2_DM260_Result_Data_64_bytes_1[33] := HwInputs.ST40_2_DM260_Result_Data_64_bytes_1[33];
	PlcInputs.ST40_2_DM260_Result_Data_64_bytes_1[34] := HwInputs.ST40_2_DM260_Result_Data_64_bytes_1[34];
	PlcInputs.ST40_2_DM260_Result_Data_64_bytes_1[35] := HwInputs.ST40_2_DM260_Result_Data_64_bytes_1[35];
	PlcInputs.ST40_2_DM260_Result_Data_64_bytes_1[36] := HwInputs.ST40_2_DM260_Result_Data_64_bytes_1[36];
	PlcInputs.ST40_2_DM260_Result_Data_64_bytes_1[37] := HwInputs.ST40_2_DM260_Result_Data_64_bytes_1[37];
	PlcInputs.ST40_2_DM260_Result_Data_64_bytes_1[38] := HwInputs.ST40_2_DM260_Result_Data_64_bytes_1[38];
	PlcInputs.ST40_2_DM260_Result_Data_64_bytes_1[39] := HwInputs.ST40_2_DM260_Result_Data_64_bytes_1[39];
	PlcInputs.ST40_2_DM260_Result_Data_64_bytes_1[40] := HwInputs.ST40_2_DM260_Result_Data_64_bytes_1[40];
	PlcInputs.ST40_2_DM260_Result_Data_64_bytes_1[41] := HwInputs.ST40_2_DM260_Result_Data_64_bytes_1[41];
	PlcInputs.ST40_2_DM260_Result_Data_64_bytes_1[42] := HwInputs.ST40_2_DM260_Result_Data_64_bytes_1[42];
	PlcInputs.ST40_2_DM260_Result_Data_64_bytes_1[43] := HwInputs.ST40_2_DM260_Result_Data_64_bytes_1[43];
	PlcInputs.ST40_2_DM260_Result_Data_64_bytes_1[44] := HwInputs.ST40_2_DM260_Result_Data_64_bytes_1[44];
	PlcInputs.ST40_2_DM260_Result_Data_64_bytes_1[45] := HwInputs.ST40_2_DM260_Result_Data_64_bytes_1[45];
	PlcInputs.ST40_2_DM260_Result_Data_64_bytes_1[46] := HwInputs.ST40_2_DM260_Result_Data_64_bytes_1[46];
	PlcInputs.ST40_2_DM260_Result_Data_64_bytes_1[47] := HwInputs.ST40_2_DM260_Result_Data_64_bytes_1[47];
	PlcInputs.ST40_2_DM260_Result_Data_64_bytes_1[48] := HwInputs.ST40_2_DM260_Result_Data_64_bytes_1[48];
	PlcInputs.ST40_2_DM260_Result_Data_64_bytes_1[49] := HwInputs.ST40_2_DM260_Result_Data_64_bytes_1[49];
	PlcInputs.ST40_2_DM260_Result_Data_64_bytes_1[50] := HwInputs.ST40_2_DM260_Result_Data_64_bytes_1[50];
	PlcInputs.ST40_2_DM260_Result_Data_64_bytes_1[51] := HwInputs.ST40_2_DM260_Result_Data_64_bytes_1[51];
	PlcInputs.ST40_2_DM260_Result_Data_64_bytes_1[52] := HwInputs.ST40_2_DM260_Result_Data_64_bytes_1[52];
	PlcInputs.ST40_2_DM260_Result_Data_64_bytes_1[53] := HwInputs.ST40_2_DM260_Result_Data_64_bytes_1[53];
	PlcInputs.ST40_2_DM260_Result_Data_64_bytes_1[54] := HwInputs.ST40_2_DM260_Result_Data_64_bytes_1[54];
	PlcInputs.ST40_2_DM260_Result_Data_64_bytes_1[55] := HwInputs.ST40_2_DM260_Result_Data_64_bytes_1[55];
	PlcInputs.ST40_2_DM260_Result_Data_64_bytes_1[56] := HwInputs.ST40_2_DM260_Result_Data_64_bytes_1[56];
	PlcInputs.ST40_2_DM260_Result_Data_64_bytes_1[57] := HwInputs.ST40_2_DM260_Result_Data_64_bytes_1[57];
	PlcInputs.ST40_2_DM260_Result_Data_64_bytes_1[58] := HwInputs.ST40_2_DM260_Result_Data_64_bytes_1[58];
	PlcInputs.ST40_2_DM260_Result_Data_64_bytes_1[59] := HwInputs.ST40_2_DM260_Result_Data_64_bytes_1[59];
	PlcInputs.ST40_2_DM260_Result_Data_64_bytes_1[60] := HwInputs.ST40_2_DM260_Result_Data_64_bytes_1[60];
	PlcInputs.ST40_2_DM260_Result_Data_64_bytes_1[61] := HwInputs.ST40_2_DM260_Result_Data_64_bytes_1[61];
	PlcInputs.ST40_2_DM260_Result_Data_64_bytes_1[62] := HwInputs.ST40_2_DM260_Result_Data_64_bytes_1[62];
	PlcInputs.ST40_2_DM260_Result_Data_64_bytes_1[63] := HwInputs.ST40_2_DM260_Result_Data_64_bytes_1[63];
	PlcInputs.ST40_2_DM260_Result_Data_64_bytes_1[64] := HwInputs.ST40_2_DM260_Result_Data_64_bytes_1[64];
	PlcInputs.ST40_2_DM260_Result_Data_64_bytes_1[65] := HwInputs.ST40_2_DM260_Result_Data_64_bytes_1[65];
	PlcInputs.ST40_2_DM260_Result_Data_64_bytes_1[66] := HwInputs.ST40_2_DM260_Result_Data_64_bytes_1[66];
	PlcInputs.ST40_2_DM260_Result_Data_64_bytes_1[67] := HwInputs.ST40_2_DM260_Result_Data_64_bytes_1[67];
	PlcInputs.ST40_2_DM260_Result_Data_64_bytes_1[68] := HwInputs.ST40_2_DM260_Result_Data_64_bytes_1[68];
	PlcInputs.ST40_2_DM260_Result_Data_64_bytes_1[69] := HwInputs.ST40_2_DM260_Result_Data_64_bytes_1[69];
	PlcInputs.ST40_2_DM260_Result_Data_64_bytes_1[70] := HwInputs.ST40_2_DM260_Result_Data_64_bytes_1[70];
	PlcInputs.ST40_2_DM260_Result_Data_64_bytes_1[71] := HwInputs.ST40_2_DM260_Result_Data_64_bytes_1[71];
	PlcInputs.ST40_3_DM260_Acquisition_Status_1[0] := HwInputs.ST40_3_DM260_Acquisition_Status_1[0];
	PlcInputs.ST40_3_DM260_Acquisition_Status_1[1] := HwInputs.ST40_3_DM260_Acquisition_Status_1[1];
	PlcInputs.ST40_3_DM260_Acquisition_Status_1[2] := HwInputs.ST40_3_DM260_Acquisition_Status_1[2];
	PlcInputs.ST40_3_DM260_Results_Status_1 := HwInputs.ST40_3_DM260_Results_Status_1;
	PlcInputs.ST40_3_DM260_Soft_Event_Control_1 := HwInputs.ST40_3_DM260_Soft_Event_Control_1;
	PlcInputs.ST40_3_DM260_Result_Data_64_bytes_1[0] := HwInputs.ST40_3_DM260_Result_Data_64_bytes_1[0];
	PlcInputs.ST40_3_DM260_Result_Data_64_bytes_1[1] := HwInputs.ST40_3_DM260_Result_Data_64_bytes_1[1];
	PlcInputs.ST40_3_DM260_Result_Data_64_bytes_1[2] := HwInputs.ST40_3_DM260_Result_Data_64_bytes_1[2];
	PlcInputs.ST40_3_DM260_Result_Data_64_bytes_1[3] := HwInputs.ST40_3_DM260_Result_Data_64_bytes_1[3];
	PlcInputs.ST40_3_DM260_Result_Data_64_bytes_1[4] := HwInputs.ST40_3_DM260_Result_Data_64_bytes_1[4];
	PlcInputs.ST40_3_DM260_Result_Data_64_bytes_1[5] := HwInputs.ST40_3_DM260_Result_Data_64_bytes_1[5];
	PlcInputs.ST40_3_DM260_Result_Data_64_bytes_1[6] := HwInputs.ST40_3_DM260_Result_Data_64_bytes_1[6];
	PlcInputs.ST40_3_DM260_Result_Data_64_bytes_1[7] := HwInputs.ST40_3_DM260_Result_Data_64_bytes_1[7];
	PlcInputs.ST40_3_DM260_Result_Data_64_bytes_1[8] := HwInputs.ST40_3_DM260_Result_Data_64_bytes_1[8];
	PlcInputs.ST40_3_DM260_Result_Data_64_bytes_1[9] := HwInputs.ST40_3_DM260_Result_Data_64_bytes_1[9];
	PlcInputs.ST40_3_DM260_Result_Data_64_bytes_1[10] := HwInputs.ST40_3_DM260_Result_Data_64_bytes_1[10];
	PlcInputs.ST40_3_DM260_Result_Data_64_bytes_1[11] := HwInputs.ST40_3_DM260_Result_Data_64_bytes_1[11];
	PlcInputs.ST40_3_DM260_Result_Data_64_bytes_1[12] := HwInputs.ST40_3_DM260_Result_Data_64_bytes_1[12];
	PlcInputs.ST40_3_DM260_Result_Data_64_bytes_1[13] := HwInputs.ST40_3_DM260_Result_Data_64_bytes_1[13];
	PlcInputs.ST40_3_DM260_Result_Data_64_bytes_1[14] := HwInputs.ST40_3_DM260_Result_Data_64_bytes_1[14];
	PlcInputs.ST40_3_DM260_Result_Data_64_bytes_1[15] := HwInputs.ST40_3_DM260_Result_Data_64_bytes_1[15];
	PlcInputs.ST40_3_DM260_Result_Data_64_bytes_1[16] := HwInputs.ST40_3_DM260_Result_Data_64_bytes_1[16];
	PlcInputs.ST40_3_DM260_Result_Data_64_bytes_1[17] := HwInputs.ST40_3_DM260_Result_Data_64_bytes_1[17];
	PlcInputs.ST40_3_DM260_Result_Data_64_bytes_1[18] := HwInputs.ST40_3_DM260_Result_Data_64_bytes_1[18];
	PlcInputs.ST40_3_DM260_Result_Data_64_bytes_1[19] := HwInputs.ST40_3_DM260_Result_Data_64_bytes_1[19];
	PlcInputs.ST40_3_DM260_Result_Data_64_bytes_1[20] := HwInputs.ST40_3_DM260_Result_Data_64_bytes_1[20];
	PlcInputs.ST40_3_DM260_Result_Data_64_bytes_1[21] := HwInputs.ST40_3_DM260_Result_Data_64_bytes_1[21];
	PlcInputs.ST40_3_DM260_Result_Data_64_bytes_1[22] := HwInputs.ST40_3_DM260_Result_Data_64_bytes_1[22];
	PlcInputs.ST40_3_DM260_Result_Data_64_bytes_1[23] := HwInputs.ST40_3_DM260_Result_Data_64_bytes_1[23];
	PlcInputs.ST40_3_DM260_Result_Data_64_bytes_1[24] := HwInputs.ST40_3_DM260_Result_Data_64_bytes_1[24];
	PlcInputs.ST40_3_DM260_Result_Data_64_bytes_1[25] := HwInputs.ST40_3_DM260_Result_Data_64_bytes_1[25];
	PlcInputs.ST40_3_DM260_Result_Data_64_bytes_1[26] := HwInputs.ST40_3_DM260_Result_Data_64_bytes_1[26];
	PlcInputs.ST40_3_DM260_Result_Data_64_bytes_1[27] := HwInputs.ST40_3_DM260_Result_Data_64_bytes_1[27];
	PlcInputs.ST40_3_DM260_Result_Data_64_bytes_1[28] := HwInputs.ST40_3_DM260_Result_Data_64_bytes_1[28];
	PlcInputs.ST40_3_DM260_Result_Data_64_bytes_1[29] := HwInputs.ST40_3_DM260_Result_Data_64_bytes_1[29];
	PlcInputs.ST40_3_DM260_Result_Data_64_bytes_1[30] := HwInputs.ST40_3_DM260_Result_Data_64_bytes_1[30];
	PlcInputs.ST40_3_DM260_Result_Data_64_bytes_1[31] := HwInputs.ST40_3_DM260_Result_Data_64_bytes_1[31];
	PlcInputs.ST40_3_DM260_Result_Data_64_bytes_1[32] := HwInputs.ST40_3_DM260_Result_Data_64_bytes_1[32];
	PlcInputs.ST40_3_DM260_Result_Data_64_bytes_1[33] := HwInputs.ST40_3_DM260_Result_Data_64_bytes_1[33];
	PlcInputs.ST40_3_DM260_Result_Data_64_bytes_1[34] := HwInputs.ST40_3_DM260_Result_Data_64_bytes_1[34];
	PlcInputs.ST40_3_DM260_Result_Data_64_bytes_1[35] := HwInputs.ST40_3_DM260_Result_Data_64_bytes_1[35];
	PlcInputs.ST40_3_DM260_Result_Data_64_bytes_1[36] := HwInputs.ST40_3_DM260_Result_Data_64_bytes_1[36];
	PlcInputs.ST40_3_DM260_Result_Data_64_bytes_1[37] := HwInputs.ST40_3_DM260_Result_Data_64_bytes_1[37];
	PlcInputs.ST40_3_DM260_Result_Data_64_bytes_1[38] := HwInputs.ST40_3_DM260_Result_Data_64_bytes_1[38];
	PlcInputs.ST40_3_DM260_Result_Data_64_bytes_1[39] := HwInputs.ST40_3_DM260_Result_Data_64_bytes_1[39];
	PlcInputs.ST40_3_DM260_Result_Data_64_bytes_1[40] := HwInputs.ST40_3_DM260_Result_Data_64_bytes_1[40];
	PlcInputs.ST40_3_DM260_Result_Data_64_bytes_1[41] := HwInputs.ST40_3_DM260_Result_Data_64_bytes_1[41];
	PlcInputs.ST40_3_DM260_Result_Data_64_bytes_1[42] := HwInputs.ST40_3_DM260_Result_Data_64_bytes_1[42];
	PlcInputs.ST40_3_DM260_Result_Data_64_bytes_1[43] := HwInputs.ST40_3_DM260_Result_Data_64_bytes_1[43];
	PlcInputs.ST40_3_DM260_Result_Data_64_bytes_1[44] := HwInputs.ST40_3_DM260_Result_Data_64_bytes_1[44];
	PlcInputs.ST40_3_DM260_Result_Data_64_bytes_1[45] := HwInputs.ST40_3_DM260_Result_Data_64_bytes_1[45];
	PlcInputs.ST40_3_DM260_Result_Data_64_bytes_1[46] := HwInputs.ST40_3_DM260_Result_Data_64_bytes_1[46];
	PlcInputs.ST40_3_DM260_Result_Data_64_bytes_1[47] := HwInputs.ST40_3_DM260_Result_Data_64_bytes_1[47];
	PlcInputs.ST40_3_DM260_Result_Data_64_bytes_1[48] := HwInputs.ST40_3_DM260_Result_Data_64_bytes_1[48];
	PlcInputs.ST40_3_DM260_Result_Data_64_bytes_1[49] := HwInputs.ST40_3_DM260_Result_Data_64_bytes_1[49];
	PlcInputs.ST40_3_DM260_Result_Data_64_bytes_1[50] := HwInputs.ST40_3_DM260_Result_Data_64_bytes_1[50];
	PlcInputs.ST40_3_DM260_Result_Data_64_bytes_1[51] := HwInputs.ST40_3_DM260_Result_Data_64_bytes_1[51];
	PlcInputs.ST40_3_DM260_Result_Data_64_bytes_1[52] := HwInputs.ST40_3_DM260_Result_Data_64_bytes_1[52];
	PlcInputs.ST40_3_DM260_Result_Data_64_bytes_1[53] := HwInputs.ST40_3_DM260_Result_Data_64_bytes_1[53];
	PlcInputs.ST40_3_DM260_Result_Data_64_bytes_1[54] := HwInputs.ST40_3_DM260_Result_Data_64_bytes_1[54];
	PlcInputs.ST40_3_DM260_Result_Data_64_bytes_1[55] := HwInputs.ST40_3_DM260_Result_Data_64_bytes_1[55];
	PlcInputs.ST40_3_DM260_Result_Data_64_bytes_1[56] := HwInputs.ST40_3_DM260_Result_Data_64_bytes_1[56];
	PlcInputs.ST40_3_DM260_Result_Data_64_bytes_1[57] := HwInputs.ST40_3_DM260_Result_Data_64_bytes_1[57];
	PlcInputs.ST40_3_DM260_Result_Data_64_bytes_1[58] := HwInputs.ST40_3_DM260_Result_Data_64_bytes_1[58];
	PlcInputs.ST40_3_DM260_Result_Data_64_bytes_1[59] := HwInputs.ST40_3_DM260_Result_Data_64_bytes_1[59];
	PlcInputs.ST40_3_DM260_Result_Data_64_bytes_1[60] := HwInputs.ST40_3_DM260_Result_Data_64_bytes_1[60];
	PlcInputs.ST40_3_DM260_Result_Data_64_bytes_1[61] := HwInputs.ST40_3_DM260_Result_Data_64_bytes_1[61];
	PlcInputs.ST40_3_DM260_Result_Data_64_bytes_1[62] := HwInputs.ST40_3_DM260_Result_Data_64_bytes_1[62];
	PlcInputs.ST40_3_DM260_Result_Data_64_bytes_1[63] := HwInputs.ST40_3_DM260_Result_Data_64_bytes_1[63];
	PlcInputs.ST40_3_DM260_Result_Data_64_bytes_1[64] := HwInputs.ST40_3_DM260_Result_Data_64_bytes_1[64];
	PlcInputs.ST40_3_DM260_Result_Data_64_bytes_1[65] := HwInputs.ST40_3_DM260_Result_Data_64_bytes_1[65];
	PlcInputs.ST40_3_DM260_Result_Data_64_bytes_1[66] := HwInputs.ST40_3_DM260_Result_Data_64_bytes_1[66];
	PlcInputs.ST40_3_DM260_Result_Data_64_bytes_1[67] := HwInputs.ST40_3_DM260_Result_Data_64_bytes_1[67];
	PlcInputs.ST40_3_DM260_Result_Data_64_bytes_1[68] := HwInputs.ST40_3_DM260_Result_Data_64_bytes_1[68];
	PlcInputs.ST40_3_DM260_Result_Data_64_bytes_1[69] := HwInputs.ST40_3_DM260_Result_Data_64_bytes_1[69];
	PlcInputs.ST40_3_DM260_Result_Data_64_bytes_1[70] := HwInputs.ST40_3_DM260_Result_Data_64_bytes_1[70];
	PlcInputs.ST40_3_DM260_Result_Data_64_bytes_1[71] := HwInputs.ST40_3_DM260_Result_Data_64_bytes_1[71];
	PlcInputs.ST40_1_DM260_Acquisition_Status_1[0] := HwInputs.ST40_1_DM260_Acquisition_Status_1[0];
	PlcInputs.ST40_1_DM260_Acquisition_Status_1[1] := HwInputs.ST40_1_DM260_Acquisition_Status_1[1];
	PlcInputs.ST40_1_DM260_Acquisition_Status_1[2] := HwInputs.ST40_1_DM260_Acquisition_Status_1[2];
	PlcInputs.ST40_1_DM260_Results_Status_1 := HwInputs.ST40_1_DM260_Results_Status_1;
	PlcInputs.ST40_1_DM260_Soft_Event_Control_1 := HwInputs.ST40_1_DM260_Soft_Event_Control_1;
	PlcInputs.ST40_1_DM260_Result_Data_64_bytes_1[0] := HwInputs.ST40_1_DM260_Result_Data_64_bytes_1[0];
	PlcInputs.ST40_1_DM260_Result_Data_64_bytes_1[1] := HwInputs.ST40_1_DM260_Result_Data_64_bytes_1[1];
	PlcInputs.ST40_1_DM260_Result_Data_64_bytes_1[2] := HwInputs.ST40_1_DM260_Result_Data_64_bytes_1[2];
	PlcInputs.ST40_1_DM260_Result_Data_64_bytes_1[3] := HwInputs.ST40_1_DM260_Result_Data_64_bytes_1[3];
	PlcInputs.ST40_1_DM260_Result_Data_64_bytes_1[4] := HwInputs.ST40_1_DM260_Result_Data_64_bytes_1[4];
	PlcInputs.ST40_1_DM260_Result_Data_64_bytes_1[5] := HwInputs.ST40_1_DM260_Result_Data_64_bytes_1[5];
	PlcInputs.ST40_1_DM260_Result_Data_64_bytes_1[6] := HwInputs.ST40_1_DM260_Result_Data_64_bytes_1[6];
	PlcInputs.ST40_1_DM260_Result_Data_64_bytes_1[7] := HwInputs.ST40_1_DM260_Result_Data_64_bytes_1[7];
	PlcInputs.ST40_1_DM260_Result_Data_64_bytes_1[8] := HwInputs.ST40_1_DM260_Result_Data_64_bytes_1[8];
	PlcInputs.ST40_1_DM260_Result_Data_64_bytes_1[9] := HwInputs.ST40_1_DM260_Result_Data_64_bytes_1[9];
	PlcInputs.ST40_1_DM260_Result_Data_64_bytes_1[10] := HwInputs.ST40_1_DM260_Result_Data_64_bytes_1[10];
	PlcInputs.ST40_1_DM260_Result_Data_64_bytes_1[11] := HwInputs.ST40_1_DM260_Result_Data_64_bytes_1[11];
	PlcInputs.ST40_1_DM260_Result_Data_64_bytes_1[12] := HwInputs.ST40_1_DM260_Result_Data_64_bytes_1[12];
	PlcInputs.ST40_1_DM260_Result_Data_64_bytes_1[13] := HwInputs.ST40_1_DM260_Result_Data_64_bytes_1[13];
	PlcInputs.ST40_1_DM260_Result_Data_64_bytes_1[14] := HwInputs.ST40_1_DM260_Result_Data_64_bytes_1[14];
	PlcInputs.ST40_1_DM260_Result_Data_64_bytes_1[15] := HwInputs.ST40_1_DM260_Result_Data_64_bytes_1[15];
	PlcInputs.ST40_1_DM260_Result_Data_64_bytes_1[16] := HwInputs.ST40_1_DM260_Result_Data_64_bytes_1[16];
	PlcInputs.ST40_1_DM260_Result_Data_64_bytes_1[17] := HwInputs.ST40_1_DM260_Result_Data_64_bytes_1[17];
	PlcInputs.ST40_1_DM260_Result_Data_64_bytes_1[18] := HwInputs.ST40_1_DM260_Result_Data_64_bytes_1[18];
	PlcInputs.ST40_1_DM260_Result_Data_64_bytes_1[19] := HwInputs.ST40_1_DM260_Result_Data_64_bytes_1[19];
	PlcInputs.ST40_1_DM260_Result_Data_64_bytes_1[20] := HwInputs.ST40_1_DM260_Result_Data_64_bytes_1[20];
	PlcInputs.ST40_1_DM260_Result_Data_64_bytes_1[21] := HwInputs.ST40_1_DM260_Result_Data_64_bytes_1[21];
	PlcInputs.ST40_1_DM260_Result_Data_64_bytes_1[22] := HwInputs.ST40_1_DM260_Result_Data_64_bytes_1[22];
	PlcInputs.ST40_1_DM260_Result_Data_64_bytes_1[23] := HwInputs.ST40_1_DM260_Result_Data_64_bytes_1[23];
	PlcInputs.ST40_1_DM260_Result_Data_64_bytes_1[24] := HwInputs.ST40_1_DM260_Result_Data_64_bytes_1[24];
	PlcInputs.ST40_1_DM260_Result_Data_64_bytes_1[25] := HwInputs.ST40_1_DM260_Result_Data_64_bytes_1[25];
	PlcInputs.ST40_1_DM260_Result_Data_64_bytes_1[26] := HwInputs.ST40_1_DM260_Result_Data_64_bytes_1[26];
	PlcInputs.ST40_1_DM260_Result_Data_64_bytes_1[27] := HwInputs.ST40_1_DM260_Result_Data_64_bytes_1[27];
	PlcInputs.ST40_1_DM260_Result_Data_64_bytes_1[28] := HwInputs.ST40_1_DM260_Result_Data_64_bytes_1[28];
	PlcInputs.ST40_1_DM260_Result_Data_64_bytes_1[29] := HwInputs.ST40_1_DM260_Result_Data_64_bytes_1[29];
	PlcInputs.ST40_1_DM260_Result_Data_64_bytes_1[30] := HwInputs.ST40_1_DM260_Result_Data_64_bytes_1[30];
	PlcInputs.ST40_1_DM260_Result_Data_64_bytes_1[31] := HwInputs.ST40_1_DM260_Result_Data_64_bytes_1[31];
	PlcInputs.ST40_1_DM260_Result_Data_64_bytes_1[32] := HwInputs.ST40_1_DM260_Result_Data_64_bytes_1[32];
	PlcInputs.ST40_1_DM260_Result_Data_64_bytes_1[33] := HwInputs.ST40_1_DM260_Result_Data_64_bytes_1[33];
	PlcInputs.ST40_1_DM260_Result_Data_64_bytes_1[34] := HwInputs.ST40_1_DM260_Result_Data_64_bytes_1[34];
	PlcInputs.ST40_1_DM260_Result_Data_64_bytes_1[35] := HwInputs.ST40_1_DM260_Result_Data_64_bytes_1[35];
	PlcInputs.ST40_1_DM260_Result_Data_64_bytes_1[36] := HwInputs.ST40_1_DM260_Result_Data_64_bytes_1[36];
	PlcInputs.ST40_1_DM260_Result_Data_64_bytes_1[37] := HwInputs.ST40_1_DM260_Result_Data_64_bytes_1[37];
	PlcInputs.ST40_1_DM260_Result_Data_64_bytes_1[38] := HwInputs.ST40_1_DM260_Result_Data_64_bytes_1[38];
	PlcInputs.ST40_1_DM260_Result_Data_64_bytes_1[39] := HwInputs.ST40_1_DM260_Result_Data_64_bytes_1[39];
	PlcInputs.ST40_1_DM260_Result_Data_64_bytes_1[40] := HwInputs.ST40_1_DM260_Result_Data_64_bytes_1[40];
	PlcInputs.ST40_1_DM260_Result_Data_64_bytes_1[41] := HwInputs.ST40_1_DM260_Result_Data_64_bytes_1[41];
	PlcInputs.ST40_1_DM260_Result_Data_64_bytes_1[42] := HwInputs.ST40_1_DM260_Result_Data_64_bytes_1[42];
	PlcInputs.ST40_1_DM260_Result_Data_64_bytes_1[43] := HwInputs.ST40_1_DM260_Result_Data_64_bytes_1[43];
	PlcInputs.ST40_1_DM260_Result_Data_64_bytes_1[44] := HwInputs.ST40_1_DM260_Result_Data_64_bytes_1[44];
	PlcInputs.ST40_1_DM260_Result_Data_64_bytes_1[45] := HwInputs.ST40_1_DM260_Result_Data_64_bytes_1[45];
	PlcInputs.ST40_1_DM260_Result_Data_64_bytes_1[46] := HwInputs.ST40_1_DM260_Result_Data_64_bytes_1[46];
	PlcInputs.ST40_1_DM260_Result_Data_64_bytes_1[47] := HwInputs.ST40_1_DM260_Result_Data_64_bytes_1[47];
	PlcInputs.ST40_1_DM260_Result_Data_64_bytes_1[48] := HwInputs.ST40_1_DM260_Result_Data_64_bytes_1[48];
	PlcInputs.ST40_1_DM260_Result_Data_64_bytes_1[49] := HwInputs.ST40_1_DM260_Result_Data_64_bytes_1[49];
	PlcInputs.ST40_1_DM260_Result_Data_64_bytes_1[50] := HwInputs.ST40_1_DM260_Result_Data_64_bytes_1[50];
	PlcInputs.ST40_1_DM260_Result_Data_64_bytes_1[51] := HwInputs.ST40_1_DM260_Result_Data_64_bytes_1[51];
	PlcInputs.ST40_1_DM260_Result_Data_64_bytes_1[52] := HwInputs.ST40_1_DM260_Result_Data_64_bytes_1[52];
	PlcInputs.ST40_1_DM260_Result_Data_64_bytes_1[53] := HwInputs.ST40_1_DM260_Result_Data_64_bytes_1[53];
	PlcInputs.ST40_1_DM260_Result_Data_64_bytes_1[54] := HwInputs.ST40_1_DM260_Result_Data_64_bytes_1[54];
	PlcInputs.ST40_1_DM260_Result_Data_64_bytes_1[55] := HwInputs.ST40_1_DM260_Result_Data_64_bytes_1[55];
	PlcInputs.ST40_1_DM260_Result_Data_64_bytes_1[56] := HwInputs.ST40_1_DM260_Result_Data_64_bytes_1[56];
	PlcInputs.ST40_1_DM260_Result_Data_64_bytes_1[57] := HwInputs.ST40_1_DM260_Result_Data_64_bytes_1[57];
	PlcInputs.ST40_1_DM260_Result_Data_64_bytes_1[58] := HwInputs.ST40_1_DM260_Result_Data_64_bytes_1[58];
	PlcInputs.ST40_1_DM260_Result_Data_64_bytes_1[59] := HwInputs.ST40_1_DM260_Result_Data_64_bytes_1[59];
	PlcInputs.ST40_1_DM260_Result_Data_64_bytes_1[60] := HwInputs.ST40_1_DM260_Result_Data_64_bytes_1[60];
	PlcInputs.ST40_1_DM260_Result_Data_64_bytes_1[61] := HwInputs.ST40_1_DM260_Result_Data_64_bytes_1[61];
	PlcInputs.ST40_1_DM260_Result_Data_64_bytes_1[62] := HwInputs.ST40_1_DM260_Result_Data_64_bytes_1[62];
	PlcInputs.ST40_1_DM260_Result_Data_64_bytes_1[63] := HwInputs.ST40_1_DM260_Result_Data_64_bytes_1[63];
	PlcInputs.ST40_1_DM260_Result_Data_64_bytes_1[64] := HwInputs.ST40_1_DM260_Result_Data_64_bytes_1[64];
	PlcInputs.ST40_1_DM260_Result_Data_64_bytes_1[65] := HwInputs.ST40_1_DM260_Result_Data_64_bytes_1[65];
	PlcInputs.ST40_1_DM260_Result_Data_64_bytes_1[66] := HwInputs.ST40_1_DM260_Result_Data_64_bytes_1[66];
	PlcInputs.ST40_1_DM260_Result_Data_64_bytes_1[67] := HwInputs.ST40_1_DM260_Result_Data_64_bytes_1[67];
	PlcInputs.ST40_1_DM260_Result_Data_64_bytes_1[68] := HwInputs.ST40_1_DM260_Result_Data_64_bytes_1[68];
	PlcInputs.ST40_1_DM260_Result_Data_64_bytes_1[69] := HwInputs.ST40_1_DM260_Result_Data_64_bytes_1[69];
	PlcInputs.ST40_1_DM260_Result_Data_64_bytes_1[70] := HwInputs.ST40_1_DM260_Result_Data_64_bytes_1[70];
	PlcInputs.ST40_1_DM260_Result_Data_64_bytes_1[71] := HwInputs.ST40_1_DM260_Result_Data_64_bytes_1[71];
	PlcInputs.ST40_2_CMMT_2GF2_Promess_DO_SERVO_1_Siemens_telegram_111_PZD_12_12[0] := HwInputs.ST40_2_CMMT_2GF2_Promess_DO_SERVO_1_Siemens_telegram_111_PZD_12_12[0];
	PlcInputs.ST40_2_CMMT_2GF2_Promess_DO_SERVO_1_Siemens_telegram_111_PZD_12_12[1] := HwInputs.ST40_2_CMMT_2GF2_Promess_DO_SERVO_1_Siemens_telegram_111_PZD_12_12[1];
	PlcInputs.ST40_2_CMMT_2GF2_Promess_DO_SERVO_1_Siemens_telegram_111_PZD_12_12[2] := HwInputs.ST40_2_CMMT_2GF2_Promess_DO_SERVO_1_Siemens_telegram_111_PZD_12_12[2];
	PlcInputs.ST40_2_CMMT_2GF2_Promess_DO_SERVO_1_Siemens_telegram_111_PZD_12_12[3] := HwInputs.ST40_2_CMMT_2GF2_Promess_DO_SERVO_1_Siemens_telegram_111_PZD_12_12[3];
	PlcInputs.ST40_2_CMMT_2GF2_Promess_DO_SERVO_1_Siemens_telegram_111_PZD_12_12[4] := HwInputs.ST40_2_CMMT_2GF2_Promess_DO_SERVO_1_Siemens_telegram_111_PZD_12_12[4];
	PlcInputs.ST40_2_CMMT_2GF2_Promess_DO_SERVO_1_Siemens_telegram_111_PZD_12_12[5] := HwInputs.ST40_2_CMMT_2GF2_Promess_DO_SERVO_1_Siemens_telegram_111_PZD_12_12[5];
	PlcInputs.ST40_2_CMMT_2GF2_Promess_DO_SERVO_1_Siemens_telegram_111_PZD_12_12[6] := HwInputs.ST40_2_CMMT_2GF2_Promess_DO_SERVO_1_Siemens_telegram_111_PZD_12_12[6];
	PlcInputs.ST40_2_CMMT_2GF2_Promess_DO_SERVO_1_Siemens_telegram_111_PZD_12_12[7] := HwInputs.ST40_2_CMMT_2GF2_Promess_DO_SERVO_1_Siemens_telegram_111_PZD_12_12[7];
	PlcInputs.ST40_2_CMMT_2GF2_Promess_DO_SERVO_1_Siemens_telegram_111_PZD_12_12[8] := HwInputs.ST40_2_CMMT_2GF2_Promess_DO_SERVO_1_Siemens_telegram_111_PZD_12_12[8];
	PlcInputs.ST40_2_CMMT_2GF2_Promess_DO_SERVO_1_Siemens_telegram_111_PZD_12_12[9] := HwInputs.ST40_2_CMMT_2GF2_Promess_DO_SERVO_1_Siemens_telegram_111_PZD_12_12[9];
	PlcInputs.ST40_2_CMMT_2GF2_Promess_DO_SERVO_1_Siemens_telegram_111_PZD_12_12[10] := HwInputs.ST40_2_CMMT_2GF2_Promess_DO_SERVO_1_Siemens_telegram_111_PZD_12_12[10];
	PlcInputs.ST40_2_CMMT_2GF2_Promess_DO_SERVO_1_Siemens_telegram_111_PZD_12_12[11] := HwInputs.ST40_2_CMMT_2GF2_Promess_DO_SERVO_1_Siemens_telegram_111_PZD_12_12[11];
	PlcInputs.ST40_2_CMMT_2GF2_Promess_DO_SERVO_1_Siemens_telegram_111_PZD_12_12[12] := HwInputs.ST40_2_CMMT_2GF2_Promess_DO_SERVO_1_Siemens_telegram_111_PZD_12_12[12];
	PlcInputs.ST40_2_CMMT_2GF2_Promess_DO_SERVO_1_Siemens_telegram_111_PZD_12_12[13] := HwInputs.ST40_2_CMMT_2GF2_Promess_DO_SERVO_1_Siemens_telegram_111_PZD_12_12[13];
	PlcInputs.ST40_2_CMMT_2GF2_Promess_DO_SERVO_1_Siemens_telegram_111_PZD_12_12[14] := HwInputs.ST40_2_CMMT_2GF2_Promess_DO_SERVO_1_Siemens_telegram_111_PZD_12_12[14];
	PlcInputs.ST40_2_CMMT_2GF2_Promess_DO_SERVO_1_Siemens_telegram_111_PZD_12_12[15] := HwInputs.ST40_2_CMMT_2GF2_Promess_DO_SERVO_1_Siemens_telegram_111_PZD_12_12[15];
	PlcInputs.ST40_2_CMMT_2GF2_Promess_DO_SERVO_1_Siemens_telegram_111_PZD_12_12[16] := HwInputs.ST40_2_CMMT_2GF2_Promess_DO_SERVO_1_Siemens_telegram_111_PZD_12_12[16];
	PlcInputs.ST40_2_CMMT_2GF2_Promess_DO_SERVO_1_Siemens_telegram_111_PZD_12_12[17] := HwInputs.ST40_2_CMMT_2GF2_Promess_DO_SERVO_1_Siemens_telegram_111_PZD_12_12[17];
	PlcInputs.ST40_2_CMMT_2GF2_Promess_DO_SERVO_1_Siemens_telegram_111_PZD_12_12[18] := HwInputs.ST40_2_CMMT_2GF2_Promess_DO_SERVO_1_Siemens_telegram_111_PZD_12_12[18];
	PlcInputs.ST40_2_CMMT_2GF2_Promess_DO_SERVO_1_Siemens_telegram_111_PZD_12_12[19] := HwInputs.ST40_2_CMMT_2GF2_Promess_DO_SERVO_1_Siemens_telegram_111_PZD_12_12[19];
	PlcInputs.ST40_2_CMMT_2GF2_Promess_DO_SERVO_1_Siemens_telegram_111_PZD_12_12[20] := HwInputs.ST40_2_CMMT_2GF2_Promess_DO_SERVO_1_Siemens_telegram_111_PZD_12_12[20];
	PlcInputs.ST40_2_CMMT_2GF2_Promess_DO_SERVO_1_Siemens_telegram_111_PZD_12_12[21] := HwInputs.ST40_2_CMMT_2GF2_Promess_DO_SERVO_1_Siemens_telegram_111_PZD_12_12[21];
	PlcInputs.ST40_2_CMMT_2GF2_Promess_DO_SERVO_1_Siemens_telegram_111_PZD_12_12[22] := HwInputs.ST40_2_CMMT_2GF2_Promess_DO_SERVO_1_Siemens_telegram_111_PZD_12_12[22];
	PlcInputs.ST40_2_CMMT_2GF2_Promess_DO_SERVO_1_Siemens_telegram_111_PZD_12_12[23] := HwInputs.ST40_2_CMMT_2GF2_Promess_DO_SERVO_1_Siemens_telegram_111_PZD_12_12[23];
	PlcInputs.ST40_2_Promess_Menu_30_01_In_1 := HwInputs.ST40_2_Promess_Menu_30_01_In_1;
	PlcInputs.ST40_2_Promess_Menu_30_02_In_1 := HwInputs.ST40_2_Promess_Menu_30_02_In_1;
	PlcInputs.ST40_2_Promess_Menu_30_03_In_1 := HwInputs.ST40_2_Promess_Menu_30_03_In_1;
	PlcInputs.ST40_2_Promess_Menu_30_04_In_1 := HwInputs.ST40_2_Promess_Menu_30_04_In_1;
	PlcInputs.ST40_2_Promess_Menu_30_05_In_1 := HwInputs.ST40_2_Promess_Menu_30_05_In_1;
	PlcInputs.ST40_2_Promess_Menu_30_06_In_1 := HwInputs.ST40_2_Promess_Menu_30_06_In_1;
	PlcInputs.ST40_2_Promess_Menu_30_07_In_1 := HwInputs.ST40_2_Promess_Menu_30_07_In_1;
	PlcInputs.ST40_2_Promess_Menu_30_08_In_1 := HwInputs.ST40_2_Promess_Menu_30_08_In_1;
	PlcInputs.ST40_2_Promess_Menu_30_09_In_1 := HwInputs.ST40_2_Promess_Menu_30_09_In_1;
	PlcInputs.ST40_2_Promess_Menu_30_10_In_1 := HwInputs.ST40_2_Promess_Menu_30_10_In_1;
	PlcInputs.ST40_2_Promess_Menu_30_11_In_1 := HwInputs.ST40_2_Promess_Menu_30_11_In_1;
	PlcInputs.ST40_2_Promess_Menu_30_12_In_1 := HwInputs.ST40_2_Promess_Menu_30_12_In_1;
	PlcInputs.ST40_2_Promess_Menu_30_13_In_1 := HwInputs.ST40_2_Promess_Menu_30_13_In_1;
	PlcInputs.ST40_2_Promess_Menu_30_14_In_1 := HwInputs.ST40_2_Promess_Menu_30_14_In_1;
	PlcInputs.ST40_2_Promess_Menu_30_15_In_1 := HwInputs.ST40_2_Promess_Menu_30_15_In_1;
	PlcInputs.ST40_2_Promess_Menu_30_16_In_1 := HwInputs.ST40_2_Promess_Menu_30_16_In_1;
	PlcInputs.ST40_2_Promess_Menu_30_17_In_1 := HwInputs.ST40_2_Promess_Menu_30_17_In_1;
	PlcInputs.ST40_2_Promess_Menu_30_18_In_1 := HwInputs.ST40_2_Promess_Menu_30_18_In_1;
	PlcInputs.ST40_2_Promess_Menu_30_19_In_1 := HwInputs.ST40_2_Promess_Menu_30_19_In_1;
	PlcInputs.ST40_2_Promess_Menu_30_20_In_1 := HwInputs.ST40_2_Promess_Menu_30_20_In_1;
	PlcInputs.ST40_2_Promess_Menu_30_21_In_1 := HwInputs.ST40_2_Promess_Menu_30_21_In_1;
	PlcInputs.ST40_2_Promess_Menu_30_22_In_1 := HwInputs.ST40_2_Promess_Menu_30_22_In_1;
	PlcInputs.ST40_2_Promess_Menu_30_23_In_1 := HwInputs.ST40_2_Promess_Menu_30_23_In_1;
	PlcInputs.ST40_2_Promess_Menu_30_24_In_1 := HwInputs.ST40_2_Promess_Menu_30_24_In_1;
	PlcInputs.ST40_2_Promess_Menu_30_25_In_1 := HwInputs.ST40_2_Promess_Menu_30_25_In_1;
	PlcInputs.ST40_2_Promess_Menu_30_26_In_1 := HwInputs.ST40_2_Promess_Menu_30_26_In_1;
	PlcInputs.ST40_2_Promess_Menu_30_27_In_1 := HwInputs.ST40_2_Promess_Menu_30_27_In_1;
	PlcInputs.ST40_2_Promess_Menu_30_28_In_1 := HwInputs.ST40_2_Promess_Menu_30_28_In_1;
	PlcInputs.ST40_2_Promess_Menu_30_29_In_1 := HwInputs.ST40_2_Promess_Menu_30_29_In_1;
	PlcInputs.ST40_2_Promess_Menu_30_30_In_1 := HwInputs.ST40_2_Promess_Menu_30_30_In_1;
	PlcInputs.ST40_2_Promess_Menu_30_31_In_1 := HwInputs.ST40_2_Promess_Menu_30_31_In_1;
	PlcInputs.ST40_2_Promess_Menu_30_32_In_1 := HwInputs.ST40_2_Promess_Menu_30_32_In_1;
	PlcInputs.ST40_ET200SP_CM_4xIO_Link_1[0] := HwInputs.ST40_ET200SP_CM_4xIO_Link_1[0];
	PlcInputs.ST40_ET200SP_CM_4xIO_Link_1[1] := HwInputs.ST40_ET200SP_CM_4xIO_Link_1[1];
	PlcInputs.ST40_ET200SP_CM_4xIO_Link_1[2] := HwInputs.ST40_ET200SP_CM_4xIO_Link_1[2];
	PlcInputs.ST40_ET200SP_CM_4xIO_Link_1[3] := HwInputs.ST40_ET200SP_CM_4xIO_Link_1[3];
	PlcInputs.ST40_ET200SP_CM_4xIO_Link_1[4] := HwInputs.ST40_ET200SP_CM_4xIO_Link_1[4];
	PlcInputs.ST40_ET200SP_CM_4xIO_Link_1[5] := HwInputs.ST40_ET200SP_CM_4xIO_Link_1[5];
	PlcInputs.ST40_ET200SP_CM_4xIO_Link_1[6] := HwInputs.ST40_ET200SP_CM_4xIO_Link_1[6];
	PlcInputs.ST40_ET200SP_CM_4xIO_Link_1[7] := HwInputs.ST40_ET200SP_CM_4xIO_Link_1[7];
	PlcInputs.ST40_ET200SP_CM_4xIO_Link_1[8] := HwInputs.ST40_ET200SP_CM_4xIO_Link_1[8];
	PlcInputs.ST40_ET200SP_CM_4xIO_Link_1[9] := HwInputs.ST40_ET200SP_CM_4xIO_Link_1[9];
	PlcInputs.ST40_ET200SP_CM_4xIO_Link_1[10] := HwInputs.ST40_ET200SP_CM_4xIO_Link_1[10];
	PlcInputs.ST40_ET200SP_CM_4xIO_Link_1[11] := HwInputs.ST40_ET200SP_CM_4xIO_Link_1[11];
	PlcInputs.ST40_ET200SP_CM_4xIO_Link_1[12] := HwInputs.ST40_ET200SP_CM_4xIO_Link_1[12];
	PlcInputs.ST40_ET200SP_CM_4xIO_Link_1[13] := HwInputs.ST40_ET200SP_CM_4xIO_Link_1[13];
	PlcInputs.ST40_ET200SP_CM_4xIO_Link_1[14] := HwInputs.ST40_ET200SP_CM_4xIO_Link_1[14];
	PlcInputs.ST40_ET200SP_CM_4xIO_Link_1[15] := HwInputs.ST40_ET200SP_CM_4xIO_Link_1[15];
	PlcInputs.ST40_ET200SP_CM_4xIO_Link_1[16] := HwInputs.ST40_ET200SP_CM_4xIO_Link_1[16];
	PlcInputs.ST40_ET200SP_CM_4xIO_Link_1[17] := HwInputs.ST40_ET200SP_CM_4xIO_Link_1[17];
	PlcInputs.ST40_ET200SP_CM_4xIO_Link_1[18] := HwInputs.ST40_ET200SP_CM_4xIO_Link_1[18];
	PlcInputs.ST40_ET200SP_CM_4xIO_Link_1[19] := HwInputs.ST40_ET200SP_CM_4xIO_Link_1[19];
	PlcInputs.ST40_ET200SP_CM_4xIO_Link_1[20] := HwInputs.ST40_ET200SP_CM_4xIO_Link_1[20];
	PlcInputs.ST40_ET200SP_CM_4xIO_Link_1[21] := HwInputs.ST40_ET200SP_CM_4xIO_Link_1[21];
	PlcInputs.ST40_ET200SP_CM_4xIO_Link_1[22] := HwInputs.ST40_ET200SP_CM_4xIO_Link_1[22];
	PlcInputs.ST40_ET200SP_CM_4xIO_Link_1[23] := HwInputs.ST40_ET200SP_CM_4xIO_Link_1[23];
	PlcInputs.ST40_ET200SP_CM_4xIO_Link_1[24] := HwInputs.ST40_ET200SP_CM_4xIO_Link_1[24];
	PlcInputs.ST40_ET200SP_CM_4xIO_Link_1[25] := HwInputs.ST40_ET200SP_CM_4xIO_Link_1[25];
	PlcInputs.ST40_ET200SP_CM_4xIO_Link_1[26] := HwInputs.ST40_ET200SP_CM_4xIO_Link_1[26];
	PlcInputs.ST40_ET200SP_CM_4xIO_Link_1[27] := HwInputs.ST40_ET200SP_CM_4xIO_Link_1[27];
	PlcInputs.ST40_ET200SP_CM_4xIO_Link_1[28] := HwInputs.ST40_ET200SP_CM_4xIO_Link_1[28];
	PlcInputs.ST40_ET200SP_CM_4xIO_Link_1[29] := HwInputs.ST40_ET200SP_CM_4xIO_Link_1[29];
	PlcInputs.ST40_ET200SP_CM_4xIO_Link_1[30] := HwInputs.ST40_ET200SP_CM_4xIO_Link_1[30];
	PlcInputs.ST40_ET200SP_CM_4xIO_Link_1[31] := HwInputs.ST40_ET200SP_CM_4xIO_Link_1[31];
	PlcInputs.ST40_ET200SP_CM_4xIO_Link_2[0] := HwInputs.ST40_ET200SP_CM_4xIO_Link_2[0];
	PlcInputs.ST40_ET200SP_CM_4xIO_Link_2[1] := HwInputs.ST40_ET200SP_CM_4xIO_Link_2[1];
	PlcInputs.ST40_ET200SP_CM_4xIO_Link_2[2] := HwInputs.ST40_ET200SP_CM_4xIO_Link_2[2];
	PlcInputs.ST40_ET200SP_CM_4xIO_Link_2[3] := HwInputs.ST40_ET200SP_CM_4xIO_Link_2[3];
	PlcInputs.ST40_ET200SP_CM_4xIO_Link_2[4] := HwInputs.ST40_ET200SP_CM_4xIO_Link_2[4];
	PlcInputs.ST40_ET200SP_CM_4xIO_Link_2[5] := HwInputs.ST40_ET200SP_CM_4xIO_Link_2[5];
	PlcInputs.ST40_ET200SP_CM_4xIO_Link_2[6] := HwInputs.ST40_ET200SP_CM_4xIO_Link_2[6];
	PlcInputs.ST40_ET200SP_CM_4xIO_Link_2[7] := HwInputs.ST40_ET200SP_CM_4xIO_Link_2[7];
	PlcInputs.ST40_ET200SP_CM_4xIO_Link_2[8] := HwInputs.ST40_ET200SP_CM_4xIO_Link_2[8];
	PlcInputs.ST40_ET200SP_CM_4xIO_Link_2[9] := HwInputs.ST40_ET200SP_CM_4xIO_Link_2[9];
	PlcInputs.ST40_ET200SP_CM_4xIO_Link_2[10] := HwInputs.ST40_ET200SP_CM_4xIO_Link_2[10];
	PlcInputs.ST40_ET200SP_CM_4xIO_Link_2[11] := HwInputs.ST40_ET200SP_CM_4xIO_Link_2[11];
	PlcInputs.ST40_ET200SP_CM_4xIO_Link_2[12] := HwInputs.ST40_ET200SP_CM_4xIO_Link_2[12];
	PlcInputs.ST40_ET200SP_CM_4xIO_Link_2[13] := HwInputs.ST40_ET200SP_CM_4xIO_Link_2[13];
	PlcInputs.ST40_ET200SP_CM_4xIO_Link_2[14] := HwInputs.ST40_ET200SP_CM_4xIO_Link_2[14];
	PlcInputs.ST40_ET200SP_CM_4xIO_Link_2[15] := HwInputs.ST40_ET200SP_CM_4xIO_Link_2[15];
	PlcInputs.ST40_ET200SP_CM_4xIO_Link_2[16] := HwInputs.ST40_ET200SP_CM_4xIO_Link_2[16];
	PlcInputs.ST40_ET200SP_CM_4xIO_Link_2[17] := HwInputs.ST40_ET200SP_CM_4xIO_Link_2[17];
	PlcInputs.ST40_ET200SP_CM_4xIO_Link_2[18] := HwInputs.ST40_ET200SP_CM_4xIO_Link_2[18];
	PlcInputs.ST40_ET200SP_CM_4xIO_Link_2[19] := HwInputs.ST40_ET200SP_CM_4xIO_Link_2[19];
	PlcInputs.ST40_ET200SP_CM_4xIO_Link_2[20] := HwInputs.ST40_ET200SP_CM_4xIO_Link_2[20];
	PlcInputs.ST40_ET200SP_CM_4xIO_Link_2[21] := HwInputs.ST40_ET200SP_CM_4xIO_Link_2[21];
	PlcInputs.ST40_ET200SP_CM_4xIO_Link_2[22] := HwInputs.ST40_ET200SP_CM_4xIO_Link_2[22];
	PlcInputs.ST40_ET200SP_CM_4xIO_Link_2[23] := HwInputs.ST40_ET200SP_CM_4xIO_Link_2[23];
	PlcInputs.ST40_ET200SP_CM_4xIO_Link_2[24] := HwInputs.ST40_ET200SP_CM_4xIO_Link_2[24];
	PlcInputs.ST40_ET200SP_CM_4xIO_Link_2[25] := HwInputs.ST40_ET200SP_CM_4xIO_Link_2[25];
	PlcInputs.ST40_ET200SP_CM_4xIO_Link_2[26] := HwInputs.ST40_ET200SP_CM_4xIO_Link_2[26];
	PlcInputs.ST40_ET200SP_CM_4xIO_Link_2[27] := HwInputs.ST40_ET200SP_CM_4xIO_Link_2[27];
	PlcInputs.ST40_ET200SP_CM_4xIO_Link_2[28] := HwInputs.ST40_ET200SP_CM_4xIO_Link_2[28];
	PlcInputs.ST40_ET200SP_CM_4xIO_Link_2[29] := HwInputs.ST40_ET200SP_CM_4xIO_Link_2[29];
	PlcInputs.ST40_ET200SP_CM_4xIO_Link_2[30] := HwInputs.ST40_ET200SP_CM_4xIO_Link_2[30];
	PlcInputs.ST40_ET200SP_CM_4xIO_Link_2[31] := HwInputs.ST40_ET200SP_CM_4xIO_Link_2[31];
	PlcInputs.ST40_ET200SP_DI_8x24VDC_ST_1 := HwInputs.ST40_ET200SP_DI_8x24VDC_ST_1;
	PlcInputs.ST40_ET200SP_DI_8x24VDC_ST_2 := HwInputs.ST40_ET200SP_DI_8x24VDC_ST_2;
	PlcInputs.ST40_ET200SP_DI_16x24VDC_ST_1 := HwInputs.ST40_ET200SP_DI_16x24VDC_ST_1;
	PlcInputs.ST40_ET200SP_DI_8x24VDC_ST_3 := HwInputs.ST40_ET200SP_DI_8x24VDC_ST_3;
END_FUNCTION

(* ---- CopyOutputs.st ---- *)
FUNCTION CopyOutputs
	VAR_EXTERNAL
		HwOutputs : HwOutputs;
		PlcOutputs : PlcOutputs;
	END_VAR
	HwOutputs.ST40_2_DM260_Acquisition_Control_1 := PlcOutputs.ST40_2_DM260_Acquisition_Control_1;
	HwOutputs.ST40_2_DM260_Results_Control_1 := PlcOutputs.ST40_2_DM260_Results_Control_1;
	HwOutputs.ST40_2_DM260_Soft_Event_Control_1 := PlcOutputs.ST40_2_DM260_Soft_Event_Control_1;
	HwOutputs.ST40_2_DM260_User_Data_64_bytes_1[0] := PlcOutputs.ST40_2_DM260_User_Data_64_bytes_1[0];
	HwOutputs.ST40_2_DM260_User_Data_64_bytes_1[1] := PlcOutputs.ST40_2_DM260_User_Data_64_bytes_1[1];
	HwOutputs.ST40_2_DM260_User_Data_64_bytes_1[2] := PlcOutputs.ST40_2_DM260_User_Data_64_bytes_1[2];
	HwOutputs.ST40_2_DM260_User_Data_64_bytes_1[3] := PlcOutputs.ST40_2_DM260_User_Data_64_bytes_1[3];
	HwOutputs.ST40_2_DM260_User_Data_64_bytes_1[4] := PlcOutputs.ST40_2_DM260_User_Data_64_bytes_1[4];
	HwOutputs.ST40_2_DM260_User_Data_64_bytes_1[5] := PlcOutputs.ST40_2_DM260_User_Data_64_bytes_1[5];
	HwOutputs.ST40_2_DM260_User_Data_64_bytes_1[6] := PlcOutputs.ST40_2_DM260_User_Data_64_bytes_1[6];
	HwOutputs.ST40_2_DM260_User_Data_64_bytes_1[7] := PlcOutputs.ST40_2_DM260_User_Data_64_bytes_1[7];
	HwOutputs.ST40_2_DM260_User_Data_64_bytes_1[8] := PlcOutputs.ST40_2_DM260_User_Data_64_bytes_1[8];
	HwOutputs.ST40_2_DM260_User_Data_64_bytes_1[9] := PlcOutputs.ST40_2_DM260_User_Data_64_bytes_1[9];
	HwOutputs.ST40_2_DM260_User_Data_64_bytes_1[10] := PlcOutputs.ST40_2_DM260_User_Data_64_bytes_1[10];
	HwOutputs.ST40_2_DM260_User_Data_64_bytes_1[11] := PlcOutputs.ST40_2_DM260_User_Data_64_bytes_1[11];
	HwOutputs.ST40_2_DM260_User_Data_64_bytes_1[12] := PlcOutputs.ST40_2_DM260_User_Data_64_bytes_1[12];
	HwOutputs.ST40_2_DM260_User_Data_64_bytes_1[13] := PlcOutputs.ST40_2_DM260_User_Data_64_bytes_1[13];
	HwOutputs.ST40_2_DM260_User_Data_64_bytes_1[14] := PlcOutputs.ST40_2_DM260_User_Data_64_bytes_1[14];
	HwOutputs.ST40_2_DM260_User_Data_64_bytes_1[15] := PlcOutputs.ST40_2_DM260_User_Data_64_bytes_1[15];
	HwOutputs.ST40_2_DM260_User_Data_64_bytes_1[16] := PlcOutputs.ST40_2_DM260_User_Data_64_bytes_1[16];
	HwOutputs.ST40_2_DM260_User_Data_64_bytes_1[17] := PlcOutputs.ST40_2_DM260_User_Data_64_bytes_1[17];
	HwOutputs.ST40_2_DM260_User_Data_64_bytes_1[18] := PlcOutputs.ST40_2_DM260_User_Data_64_bytes_1[18];
	HwOutputs.ST40_2_DM260_User_Data_64_bytes_1[19] := PlcOutputs.ST40_2_DM260_User_Data_64_bytes_1[19];
	HwOutputs.ST40_2_DM260_User_Data_64_bytes_1[20] := PlcOutputs.ST40_2_DM260_User_Data_64_bytes_1[20];
	HwOutputs.ST40_2_DM260_User_Data_64_bytes_1[21] := PlcOutputs.ST40_2_DM260_User_Data_64_bytes_1[21];
	HwOutputs.ST40_2_DM260_User_Data_64_bytes_1[22] := PlcOutputs.ST40_2_DM260_User_Data_64_bytes_1[22];
	HwOutputs.ST40_2_DM260_User_Data_64_bytes_1[23] := PlcOutputs.ST40_2_DM260_User_Data_64_bytes_1[23];
	HwOutputs.ST40_2_DM260_User_Data_64_bytes_1[24] := PlcOutputs.ST40_2_DM260_User_Data_64_bytes_1[24];
	HwOutputs.ST40_2_DM260_User_Data_64_bytes_1[25] := PlcOutputs.ST40_2_DM260_User_Data_64_bytes_1[25];
	HwOutputs.ST40_2_DM260_User_Data_64_bytes_1[26] := PlcOutputs.ST40_2_DM260_User_Data_64_bytes_1[26];
	HwOutputs.ST40_2_DM260_User_Data_64_bytes_1[27] := PlcOutputs.ST40_2_DM260_User_Data_64_bytes_1[27];
	HwOutputs.ST40_2_DM260_User_Data_64_bytes_1[28] := PlcOutputs.ST40_2_DM260_User_Data_64_bytes_1[28];
	HwOutputs.ST40_2_DM260_User_Data_64_bytes_1[29] := PlcOutputs.ST40_2_DM260_User_Data_64_bytes_1[29];
	HwOutputs.ST40_2_DM260_User_Data_64_bytes_1[30] := PlcOutputs.ST40_2_DM260_User_Data_64_bytes_1[30];
	HwOutputs.ST40_2_DM260_User_Data_64_bytes_1[31] := PlcOutputs.ST40_2_DM260_User_Data_64_bytes_1[31];
	HwOutputs.ST40_2_DM260_User_Data_64_bytes_1[32] := PlcOutputs.ST40_2_DM260_User_Data_64_bytes_1[32];
	HwOutputs.ST40_2_DM260_User_Data_64_bytes_1[33] := PlcOutputs.ST40_2_DM260_User_Data_64_bytes_1[33];
	HwOutputs.ST40_2_DM260_User_Data_64_bytes_1[34] := PlcOutputs.ST40_2_DM260_User_Data_64_bytes_1[34];
	HwOutputs.ST40_2_DM260_User_Data_64_bytes_1[35] := PlcOutputs.ST40_2_DM260_User_Data_64_bytes_1[35];
	HwOutputs.ST40_2_DM260_User_Data_64_bytes_1[36] := PlcOutputs.ST40_2_DM260_User_Data_64_bytes_1[36];
	HwOutputs.ST40_2_DM260_User_Data_64_bytes_1[37] := PlcOutputs.ST40_2_DM260_User_Data_64_bytes_1[37];
	HwOutputs.ST40_2_DM260_User_Data_64_bytes_1[38] := PlcOutputs.ST40_2_DM260_User_Data_64_bytes_1[38];
	HwOutputs.ST40_2_DM260_User_Data_64_bytes_1[39] := PlcOutputs.ST40_2_DM260_User_Data_64_bytes_1[39];
	HwOutputs.ST40_2_DM260_User_Data_64_bytes_1[40] := PlcOutputs.ST40_2_DM260_User_Data_64_bytes_1[40];
	HwOutputs.ST40_2_DM260_User_Data_64_bytes_1[41] := PlcOutputs.ST40_2_DM260_User_Data_64_bytes_1[41];
	HwOutputs.ST40_2_DM260_User_Data_64_bytes_1[42] := PlcOutputs.ST40_2_DM260_User_Data_64_bytes_1[42];
	HwOutputs.ST40_2_DM260_User_Data_64_bytes_1[43] := PlcOutputs.ST40_2_DM260_User_Data_64_bytes_1[43];
	HwOutputs.ST40_2_DM260_User_Data_64_bytes_1[44] := PlcOutputs.ST40_2_DM260_User_Data_64_bytes_1[44];
	HwOutputs.ST40_2_DM260_User_Data_64_bytes_1[45] := PlcOutputs.ST40_2_DM260_User_Data_64_bytes_1[45];
	HwOutputs.ST40_2_DM260_User_Data_64_bytes_1[46] := PlcOutputs.ST40_2_DM260_User_Data_64_bytes_1[46];
	HwOutputs.ST40_2_DM260_User_Data_64_bytes_1[47] := PlcOutputs.ST40_2_DM260_User_Data_64_bytes_1[47];
	HwOutputs.ST40_2_DM260_User_Data_64_bytes_1[48] := PlcOutputs.ST40_2_DM260_User_Data_64_bytes_1[48];
	HwOutputs.ST40_2_DM260_User_Data_64_bytes_1[49] := PlcOutputs.ST40_2_DM260_User_Data_64_bytes_1[49];
	HwOutputs.ST40_2_DM260_User_Data_64_bytes_1[50] := PlcOutputs.ST40_2_DM260_User_Data_64_bytes_1[50];
	HwOutputs.ST40_2_DM260_User_Data_64_bytes_1[51] := PlcOutputs.ST40_2_DM260_User_Data_64_bytes_1[51];
	HwOutputs.ST40_2_DM260_User_Data_64_bytes_1[52] := PlcOutputs.ST40_2_DM260_User_Data_64_bytes_1[52];
	HwOutputs.ST40_2_DM260_User_Data_64_bytes_1[53] := PlcOutputs.ST40_2_DM260_User_Data_64_bytes_1[53];
	HwOutputs.ST40_2_DM260_User_Data_64_bytes_1[54] := PlcOutputs.ST40_2_DM260_User_Data_64_bytes_1[54];
	HwOutputs.ST40_2_DM260_User_Data_64_bytes_1[55] := PlcOutputs.ST40_2_DM260_User_Data_64_bytes_1[55];
	HwOutputs.ST40_2_DM260_User_Data_64_bytes_1[56] := PlcOutputs.ST40_2_DM260_User_Data_64_bytes_1[56];
	HwOutputs.ST40_2_DM260_User_Data_64_bytes_1[57] := PlcOutputs.ST40_2_DM260_User_Data_64_bytes_1[57];
	HwOutputs.ST40_2_DM260_User_Data_64_bytes_1[58] := PlcOutputs.ST40_2_DM260_User_Data_64_bytes_1[58];
	HwOutputs.ST40_2_DM260_User_Data_64_bytes_1[59] := PlcOutputs.ST40_2_DM260_User_Data_64_bytes_1[59];
	HwOutputs.ST40_2_DM260_User_Data_64_bytes_1[60] := PlcOutputs.ST40_2_DM260_User_Data_64_bytes_1[60];
	HwOutputs.ST40_2_DM260_User_Data_64_bytes_1[61] := PlcOutputs.ST40_2_DM260_User_Data_64_bytes_1[61];
	HwOutputs.ST40_2_DM260_User_Data_64_bytes_1[62] := PlcOutputs.ST40_2_DM260_User_Data_64_bytes_1[62];
	HwOutputs.ST40_2_DM260_User_Data_64_bytes_1[63] := PlcOutputs.ST40_2_DM260_User_Data_64_bytes_1[63];
	HwOutputs.ST40_2_DM260_User_Data_64_bytes_1[64] := PlcOutputs.ST40_2_DM260_User_Data_64_bytes_1[64];
	HwOutputs.ST40_2_DM260_User_Data_64_bytes_1[65] := PlcOutputs.ST40_2_DM260_User_Data_64_bytes_1[65];
	HwOutputs.ST40_2_DM260_User_Data_64_bytes_1[66] := PlcOutputs.ST40_2_DM260_User_Data_64_bytes_1[66];
	HwOutputs.ST40_2_DM260_User_Data_64_bytes_1[67] := PlcOutputs.ST40_2_DM260_User_Data_64_bytes_1[67];
	HwOutputs.ST40_3_DM260_Acquisition_Control_1 := PlcOutputs.ST40_3_DM260_Acquisition_Control_1;
	HwOutputs.ST40_3_DM260_Results_Control_1 := PlcOutputs.ST40_3_DM260_Results_Control_1;
	HwOutputs.ST40_3_DM260_Soft_Event_Control_1 := PlcOutputs.ST40_3_DM260_Soft_Event_Control_1;
	HwOutputs.ST40_3_DM260_User_Data_64_bytes_1[0] := PlcOutputs.ST40_3_DM260_User_Data_64_bytes_1[0];
	HwOutputs.ST40_3_DM260_User_Data_64_bytes_1[1] := PlcOutputs.ST40_3_DM260_User_Data_64_bytes_1[1];
	HwOutputs.ST40_3_DM260_User_Data_64_bytes_1[2] := PlcOutputs.ST40_3_DM260_User_Data_64_bytes_1[2];
	HwOutputs.ST40_3_DM260_User_Data_64_bytes_1[3] := PlcOutputs.ST40_3_DM260_User_Data_64_bytes_1[3];
	HwOutputs.ST40_3_DM260_User_Data_64_bytes_1[4] := PlcOutputs.ST40_3_DM260_User_Data_64_bytes_1[4];
	HwOutputs.ST40_3_DM260_User_Data_64_bytes_1[5] := PlcOutputs.ST40_3_DM260_User_Data_64_bytes_1[5];
	HwOutputs.ST40_3_DM260_User_Data_64_bytes_1[6] := PlcOutputs.ST40_3_DM260_User_Data_64_bytes_1[6];
	HwOutputs.ST40_3_DM260_User_Data_64_bytes_1[7] := PlcOutputs.ST40_3_DM260_User_Data_64_bytes_1[7];
	HwOutputs.ST40_3_DM260_User_Data_64_bytes_1[8] := PlcOutputs.ST40_3_DM260_User_Data_64_bytes_1[8];
	HwOutputs.ST40_3_DM260_User_Data_64_bytes_1[9] := PlcOutputs.ST40_3_DM260_User_Data_64_bytes_1[9];
	HwOutputs.ST40_3_DM260_User_Data_64_bytes_1[10] := PlcOutputs.ST40_3_DM260_User_Data_64_bytes_1[10];
	HwOutputs.ST40_3_DM260_User_Data_64_bytes_1[11] := PlcOutputs.ST40_3_DM260_User_Data_64_bytes_1[11];
	HwOutputs.ST40_3_DM260_User_Data_64_bytes_1[12] := PlcOutputs.ST40_3_DM260_User_Data_64_bytes_1[12];
	HwOutputs.ST40_3_DM260_User_Data_64_bytes_1[13] := PlcOutputs.ST40_3_DM260_User_Data_64_bytes_1[13];
	HwOutputs.ST40_3_DM260_User_Data_64_bytes_1[14] := PlcOutputs.ST40_3_DM260_User_Data_64_bytes_1[14];
	HwOutputs.ST40_3_DM260_User_Data_64_bytes_1[15] := PlcOutputs.ST40_3_DM260_User_Data_64_bytes_1[15];
	HwOutputs.ST40_3_DM260_User_Data_64_bytes_1[16] := PlcOutputs.ST40_3_DM260_User_Data_64_bytes_1[16];
	HwOutputs.ST40_3_DM260_User_Data_64_bytes_1[17] := PlcOutputs.ST40_3_DM260_User_Data_64_bytes_1[17];
	HwOutputs.ST40_3_DM260_User_Data_64_bytes_1[18] := PlcOutputs.ST40_3_DM260_User_Data_64_bytes_1[18];
	HwOutputs.ST40_3_DM260_User_Data_64_bytes_1[19] := PlcOutputs.ST40_3_DM260_User_Data_64_bytes_1[19];
	HwOutputs.ST40_3_DM260_User_Data_64_bytes_1[20] := PlcOutputs.ST40_3_DM260_User_Data_64_bytes_1[20];
	HwOutputs.ST40_3_DM260_User_Data_64_bytes_1[21] := PlcOutputs.ST40_3_DM260_User_Data_64_bytes_1[21];
	HwOutputs.ST40_3_DM260_User_Data_64_bytes_1[22] := PlcOutputs.ST40_3_DM260_User_Data_64_bytes_1[22];
	HwOutputs.ST40_3_DM260_User_Data_64_bytes_1[23] := PlcOutputs.ST40_3_DM260_User_Data_64_bytes_1[23];
	HwOutputs.ST40_3_DM260_User_Data_64_bytes_1[24] := PlcOutputs.ST40_3_DM260_User_Data_64_bytes_1[24];
	HwOutputs.ST40_3_DM260_User_Data_64_bytes_1[25] := PlcOutputs.ST40_3_DM260_User_Data_64_bytes_1[25];
	HwOutputs.ST40_3_DM260_User_Data_64_bytes_1[26] := PlcOutputs.ST40_3_DM260_User_Data_64_bytes_1[26];
	HwOutputs.ST40_3_DM260_User_Data_64_bytes_1[27] := PlcOutputs.ST40_3_DM260_User_Data_64_bytes_1[27];
	HwOutputs.ST40_3_DM260_User_Data_64_bytes_1[28] := PlcOutputs.ST40_3_DM260_User_Data_64_bytes_1[28];
	HwOutputs.ST40_3_DM260_User_Data_64_bytes_1[29] := PlcOutputs.ST40_3_DM260_User_Data_64_bytes_1[29];
	HwOutputs.ST40_3_DM260_User_Data_64_bytes_1[30] := PlcOutputs.ST40_3_DM260_User_Data_64_bytes_1[30];
	HwOutputs.ST40_3_DM260_User_Data_64_bytes_1[31] := PlcOutputs.ST40_3_DM260_User_Data_64_bytes_1[31];
	HwOutputs.ST40_3_DM260_User_Data_64_bytes_1[32] := PlcOutputs.ST40_3_DM260_User_Data_64_bytes_1[32];
	HwOutputs.ST40_3_DM260_User_Data_64_bytes_1[33] := PlcOutputs.ST40_3_DM260_User_Data_64_bytes_1[33];
	HwOutputs.ST40_3_DM260_User_Data_64_bytes_1[34] := PlcOutputs.ST40_3_DM260_User_Data_64_bytes_1[34];
	HwOutputs.ST40_3_DM260_User_Data_64_bytes_1[35] := PlcOutputs.ST40_3_DM260_User_Data_64_bytes_1[35];
	HwOutputs.ST40_3_DM260_User_Data_64_bytes_1[36] := PlcOutputs.ST40_3_DM260_User_Data_64_bytes_1[36];
	HwOutputs.ST40_3_DM260_User_Data_64_bytes_1[37] := PlcOutputs.ST40_3_DM260_User_Data_64_bytes_1[37];
	HwOutputs.ST40_3_DM260_User_Data_64_bytes_1[38] := PlcOutputs.ST40_3_DM260_User_Data_64_bytes_1[38];
	HwOutputs.ST40_3_DM260_User_Data_64_bytes_1[39] := PlcOutputs.ST40_3_DM260_User_Data_64_bytes_1[39];
	HwOutputs.ST40_3_DM260_User_Data_64_bytes_1[40] := PlcOutputs.ST40_3_DM260_User_Data_64_bytes_1[40];
	HwOutputs.ST40_3_DM260_User_Data_64_bytes_1[41] := PlcOutputs.ST40_3_DM260_User_Data_64_bytes_1[41];
	HwOutputs.ST40_3_DM260_User_Data_64_bytes_1[42] := PlcOutputs.ST40_3_DM260_User_Data_64_bytes_1[42];
	HwOutputs.ST40_3_DM260_User_Data_64_bytes_1[43] := PlcOutputs.ST40_3_DM260_User_Data_64_bytes_1[43];
	HwOutputs.ST40_3_DM260_User_Data_64_bytes_1[44] := PlcOutputs.ST40_3_DM260_User_Data_64_bytes_1[44];
	HwOutputs.ST40_3_DM260_User_Data_64_bytes_1[45] := PlcOutputs.ST40_3_DM260_User_Data_64_bytes_1[45];
	HwOutputs.ST40_3_DM260_User_Data_64_bytes_1[46] := PlcOutputs.ST40_3_DM260_User_Data_64_bytes_1[46];
	HwOutputs.ST40_3_DM260_User_Data_64_bytes_1[47] := PlcOutputs.ST40_3_DM260_User_Data_64_bytes_1[47];
	HwOutputs.ST40_3_DM260_User_Data_64_bytes_1[48] := PlcOutputs.ST40_3_DM260_User_Data_64_bytes_1[48];
	HwOutputs.ST40_3_DM260_User_Data_64_bytes_1[49] := PlcOutputs.ST40_3_DM260_User_Data_64_bytes_1[49];
	HwOutputs.ST40_3_DM260_User_Data_64_bytes_1[50] := PlcOutputs.ST40_3_DM260_User_Data_64_bytes_1[50];
	HwOutputs.ST40_3_DM260_User_Data_64_bytes_1[51] := PlcOutputs.ST40_3_DM260_User_Data_64_bytes_1[51];
	HwOutputs.ST40_3_DM260_User_Data_64_bytes_1[52] := PlcOutputs.ST40_3_DM260_User_Data_64_bytes_1[52];
	HwOutputs.ST40_3_DM260_User_Data_64_bytes_1[53] := PlcOutputs.ST40_3_DM260_User_Data_64_bytes_1[53];
	HwOutputs.ST40_3_DM260_User_Data_64_bytes_1[54] := PlcOutputs.ST40_3_DM260_User_Data_64_bytes_1[54];
	HwOutputs.ST40_3_DM260_User_Data_64_bytes_1[55] := PlcOutputs.ST40_3_DM260_User_Data_64_bytes_1[55];
	HwOutputs.ST40_3_DM260_User_Data_64_bytes_1[56] := PlcOutputs.ST40_3_DM260_User_Data_64_bytes_1[56];
	HwOutputs.ST40_3_DM260_User_Data_64_bytes_1[57] := PlcOutputs.ST40_3_DM260_User_Data_64_bytes_1[57];
	HwOutputs.ST40_3_DM260_User_Data_64_bytes_1[58] := PlcOutputs.ST40_3_DM260_User_Data_64_bytes_1[58];
	HwOutputs.ST40_3_DM260_User_Data_64_bytes_1[59] := PlcOutputs.ST40_3_DM260_User_Data_64_bytes_1[59];
	HwOutputs.ST40_3_DM260_User_Data_64_bytes_1[60] := PlcOutputs.ST40_3_DM260_User_Data_64_bytes_1[60];
	HwOutputs.ST40_3_DM260_User_Data_64_bytes_1[61] := PlcOutputs.ST40_3_DM260_User_Data_64_bytes_1[61];
	HwOutputs.ST40_3_DM260_User_Data_64_bytes_1[62] := PlcOutputs.ST40_3_DM260_User_Data_64_bytes_1[62];
	HwOutputs.ST40_3_DM260_User_Data_64_bytes_1[63] := PlcOutputs.ST40_3_DM260_User_Data_64_bytes_1[63];
	HwOutputs.ST40_3_DM260_User_Data_64_bytes_1[64] := PlcOutputs.ST40_3_DM260_User_Data_64_bytes_1[64];
	HwOutputs.ST40_3_DM260_User_Data_64_bytes_1[65] := PlcOutputs.ST40_3_DM260_User_Data_64_bytes_1[65];
	HwOutputs.ST40_3_DM260_User_Data_64_bytes_1[66] := PlcOutputs.ST40_3_DM260_User_Data_64_bytes_1[66];
	HwOutputs.ST40_3_DM260_User_Data_64_bytes_1[67] := PlcOutputs.ST40_3_DM260_User_Data_64_bytes_1[67];
	HwOutputs.ST40_1_DM260_Acquisition_Control_1 := PlcOutputs.ST40_1_DM260_Acquisition_Control_1;
	HwOutputs.ST40_1_DM260_Results_Control_1 := PlcOutputs.ST40_1_DM260_Results_Control_1;
	HwOutputs.ST40_1_DM260_Soft_Event_Control_1 := PlcOutputs.ST40_1_DM260_Soft_Event_Control_1;
	HwOutputs.ST40_1_DM260_User_Data_64_bytes_1[0] := PlcOutputs.ST40_1_DM260_User_Data_64_bytes_1[0];
	HwOutputs.ST40_1_DM260_User_Data_64_bytes_1[1] := PlcOutputs.ST40_1_DM260_User_Data_64_bytes_1[1];
	HwOutputs.ST40_1_DM260_User_Data_64_bytes_1[2] := PlcOutputs.ST40_1_DM260_User_Data_64_bytes_1[2];
	HwOutputs.ST40_1_DM260_User_Data_64_bytes_1[3] := PlcOutputs.ST40_1_DM260_User_Data_64_bytes_1[3];
	HwOutputs.ST40_1_DM260_User_Data_64_bytes_1[4] := PlcOutputs.ST40_1_DM260_User_Data_64_bytes_1[4];
	HwOutputs.ST40_1_DM260_User_Data_64_bytes_1[5] := PlcOutputs.ST40_1_DM260_User_Data_64_bytes_1[5];
	HwOutputs.ST40_1_DM260_User_Data_64_bytes_1[6] := PlcOutputs.ST40_1_DM260_User_Data_64_bytes_1[6];
	HwOutputs.ST40_1_DM260_User_Data_64_bytes_1[7] := PlcOutputs.ST40_1_DM260_User_Data_64_bytes_1[7];
	HwOutputs.ST40_1_DM260_User_Data_64_bytes_1[8] := PlcOutputs.ST40_1_DM260_User_Data_64_bytes_1[8];
	HwOutputs.ST40_1_DM260_User_Data_64_bytes_1[9] := PlcOutputs.ST40_1_DM260_User_Data_64_bytes_1[9];
	HwOutputs.ST40_1_DM260_User_Data_64_bytes_1[10] := PlcOutputs.ST40_1_DM260_User_Data_64_bytes_1[10];
	HwOutputs.ST40_1_DM260_User_Data_64_bytes_1[11] := PlcOutputs.ST40_1_DM260_User_Data_64_bytes_1[11];
	HwOutputs.ST40_1_DM260_User_Data_64_bytes_1[12] := PlcOutputs.ST40_1_DM260_User_Data_64_bytes_1[12];
	HwOutputs.ST40_1_DM260_User_Data_64_bytes_1[13] := PlcOutputs.ST40_1_DM260_User_Data_64_bytes_1[13];
	HwOutputs.ST40_1_DM260_User_Data_64_bytes_1[14] := PlcOutputs.ST40_1_DM260_User_Data_64_bytes_1[14];
	HwOutputs.ST40_1_DM260_User_Data_64_bytes_1[15] := PlcOutputs.ST40_1_DM260_User_Data_64_bytes_1[15];
	HwOutputs.ST40_1_DM260_User_Data_64_bytes_1[16] := PlcOutputs.ST40_1_DM260_User_Data_64_bytes_1[16];
	HwOutputs.ST40_1_DM260_User_Data_64_bytes_1[17] := PlcOutputs.ST40_1_DM260_User_Data_64_bytes_1[17];
	HwOutputs.ST40_1_DM260_User_Data_64_bytes_1[18] := PlcOutputs.ST40_1_DM260_User_Data_64_bytes_1[18];
	HwOutputs.ST40_1_DM260_User_Data_64_bytes_1[19] := PlcOutputs.ST40_1_DM260_User_Data_64_bytes_1[19];
	HwOutputs.ST40_1_DM260_User_Data_64_bytes_1[20] := PlcOutputs.ST40_1_DM260_User_Data_64_bytes_1[20];
	HwOutputs.ST40_1_DM260_User_Data_64_bytes_1[21] := PlcOutputs.ST40_1_DM260_User_Data_64_bytes_1[21];
	HwOutputs.ST40_1_DM260_User_Data_64_bytes_1[22] := PlcOutputs.ST40_1_DM260_User_Data_64_bytes_1[22];
	HwOutputs.ST40_1_DM260_User_Data_64_bytes_1[23] := PlcOutputs.ST40_1_DM260_User_Data_64_bytes_1[23];
	HwOutputs.ST40_1_DM260_User_Data_64_bytes_1[24] := PlcOutputs.ST40_1_DM260_User_Data_64_bytes_1[24];
	HwOutputs.ST40_1_DM260_User_Data_64_bytes_1[25] := PlcOutputs.ST40_1_DM260_User_Data_64_bytes_1[25];
	HwOutputs.ST40_1_DM260_User_Data_64_bytes_1[26] := PlcOutputs.ST40_1_DM260_User_Data_64_bytes_1[26];
	HwOutputs.ST40_1_DM260_User_Data_64_bytes_1[27] := PlcOutputs.ST40_1_DM260_User_Data_64_bytes_1[27];
	HwOutputs.ST40_1_DM260_User_Data_64_bytes_1[28] := PlcOutputs.ST40_1_DM260_User_Data_64_bytes_1[28];
	HwOutputs.ST40_1_DM260_User_Data_64_bytes_1[29] := PlcOutputs.ST40_1_DM260_User_Data_64_bytes_1[29];
	HwOutputs.ST40_1_DM260_User_Data_64_bytes_1[30] := PlcOutputs.ST40_1_DM260_User_Data_64_bytes_1[30];
	HwOutputs.ST40_1_DM260_User_Data_64_bytes_1[31] := PlcOutputs.ST40_1_DM260_User_Data_64_bytes_1[31];
	HwOutputs.ST40_1_DM260_User_Data_64_bytes_1[32] := PlcOutputs.ST40_1_DM260_User_Data_64_bytes_1[32];
	HwOutputs.ST40_1_DM260_User_Data_64_bytes_1[33] := PlcOutputs.ST40_1_DM260_User_Data_64_bytes_1[33];
	HwOutputs.ST40_1_DM260_User_Data_64_bytes_1[34] := PlcOutputs.ST40_1_DM260_User_Data_64_bytes_1[34];
	HwOutputs.ST40_1_DM260_User_Data_64_bytes_1[35] := PlcOutputs.ST40_1_DM260_User_Data_64_bytes_1[35];
	HwOutputs.ST40_1_DM260_User_Data_64_bytes_1[36] := PlcOutputs.ST40_1_DM260_User_Data_64_bytes_1[36];
	HwOutputs.ST40_1_DM260_User_Data_64_bytes_1[37] := PlcOutputs.ST40_1_DM260_User_Data_64_bytes_1[37];
	HwOutputs.ST40_1_DM260_User_Data_64_bytes_1[38] := PlcOutputs.ST40_1_DM260_User_Data_64_bytes_1[38];
	HwOutputs.ST40_1_DM260_User_Data_64_bytes_1[39] := PlcOutputs.ST40_1_DM260_User_Data_64_bytes_1[39];
	HwOutputs.ST40_1_DM260_User_Data_64_bytes_1[40] := PlcOutputs.ST40_1_DM260_User_Data_64_bytes_1[40];
	HwOutputs.ST40_1_DM260_User_Data_64_bytes_1[41] := PlcOutputs.ST40_1_DM260_User_Data_64_bytes_1[41];
	HwOutputs.ST40_1_DM260_User_Data_64_bytes_1[42] := PlcOutputs.ST40_1_DM260_User_Data_64_bytes_1[42];
	HwOutputs.ST40_1_DM260_User_Data_64_bytes_1[43] := PlcOutputs.ST40_1_DM260_User_Data_64_bytes_1[43];
	HwOutputs.ST40_1_DM260_User_Data_64_bytes_1[44] := PlcOutputs.ST40_1_DM260_User_Data_64_bytes_1[44];
	HwOutputs.ST40_1_DM260_User_Data_64_bytes_1[45] := PlcOutputs.ST40_1_DM260_User_Data_64_bytes_1[45];
	HwOutputs.ST40_1_DM260_User_Data_64_bytes_1[46] := PlcOutputs.ST40_1_DM260_User_Data_64_bytes_1[46];
	HwOutputs.ST40_1_DM260_User_Data_64_bytes_1[47] := PlcOutputs.ST40_1_DM260_User_Data_64_bytes_1[47];
	HwOutputs.ST40_1_DM260_User_Data_64_bytes_1[48] := PlcOutputs.ST40_1_DM260_User_Data_64_bytes_1[48];
	HwOutputs.ST40_1_DM260_User_Data_64_bytes_1[49] := PlcOutputs.ST40_1_DM260_User_Data_64_bytes_1[49];
	HwOutputs.ST40_1_DM260_User_Data_64_bytes_1[50] := PlcOutputs.ST40_1_DM260_User_Data_64_bytes_1[50];
	HwOutputs.ST40_1_DM260_User_Data_64_bytes_1[51] := PlcOutputs.ST40_1_DM260_User_Data_64_bytes_1[51];
	HwOutputs.ST40_1_DM260_User_Data_64_bytes_1[52] := PlcOutputs.ST40_1_DM260_User_Data_64_bytes_1[52];
	HwOutputs.ST40_1_DM260_User_Data_64_bytes_1[53] := PlcOutputs.ST40_1_DM260_User_Data_64_bytes_1[53];
	HwOutputs.ST40_1_DM260_User_Data_64_bytes_1[54] := PlcOutputs.ST40_1_DM260_User_Data_64_bytes_1[54];
	HwOutputs.ST40_1_DM260_User_Data_64_bytes_1[55] := PlcOutputs.ST40_1_DM260_User_Data_64_bytes_1[55];
	HwOutputs.ST40_1_DM260_User_Data_64_bytes_1[56] := PlcOutputs.ST40_1_DM260_User_Data_64_bytes_1[56];
	HwOutputs.ST40_1_DM260_User_Data_64_bytes_1[57] := PlcOutputs.ST40_1_DM260_User_Data_64_bytes_1[57];
	HwOutputs.ST40_1_DM260_User_Data_64_bytes_1[58] := PlcOutputs.ST40_1_DM260_User_Data_64_bytes_1[58];
	HwOutputs.ST40_1_DM260_User_Data_64_bytes_1[59] := PlcOutputs.ST40_1_DM260_User_Data_64_bytes_1[59];
	HwOutputs.ST40_1_DM260_User_Data_64_bytes_1[60] := PlcOutputs.ST40_1_DM260_User_Data_64_bytes_1[60];
	HwOutputs.ST40_1_DM260_User_Data_64_bytes_1[61] := PlcOutputs.ST40_1_DM260_User_Data_64_bytes_1[61];
	HwOutputs.ST40_1_DM260_User_Data_64_bytes_1[62] := PlcOutputs.ST40_1_DM260_User_Data_64_bytes_1[62];
	HwOutputs.ST40_1_DM260_User_Data_64_bytes_1[63] := PlcOutputs.ST40_1_DM260_User_Data_64_bytes_1[63];
	HwOutputs.ST40_1_DM260_User_Data_64_bytes_1[64] := PlcOutputs.ST40_1_DM260_User_Data_64_bytes_1[64];
	HwOutputs.ST40_1_DM260_User_Data_64_bytes_1[65] := PlcOutputs.ST40_1_DM260_User_Data_64_bytes_1[65];
	HwOutputs.ST40_1_DM260_User_Data_64_bytes_1[66] := PlcOutputs.ST40_1_DM260_User_Data_64_bytes_1[66];
	HwOutputs.ST40_1_DM260_User_Data_64_bytes_1[67] := PlcOutputs.ST40_1_DM260_User_Data_64_bytes_1[67];
	HwOutputs.ST40_2_CMMT_2GF2_Promess_DO_SERVO_1_Siemens_telegram_111_PZD_12_12[0] := PlcOutputs.ST40_2_CMMT_2GF2_Promess_DO_SERVO_1_Siemens_telegram_111_PZD_12_12[0];
	HwOutputs.ST40_2_CMMT_2GF2_Promess_DO_SERVO_1_Siemens_telegram_111_PZD_12_12[1] := PlcOutputs.ST40_2_CMMT_2GF2_Promess_DO_SERVO_1_Siemens_telegram_111_PZD_12_12[1];
	HwOutputs.ST40_2_CMMT_2GF2_Promess_DO_SERVO_1_Siemens_telegram_111_PZD_12_12[2] := PlcOutputs.ST40_2_CMMT_2GF2_Promess_DO_SERVO_1_Siemens_telegram_111_PZD_12_12[2];
	HwOutputs.ST40_2_CMMT_2GF2_Promess_DO_SERVO_1_Siemens_telegram_111_PZD_12_12[3] := PlcOutputs.ST40_2_CMMT_2GF2_Promess_DO_SERVO_1_Siemens_telegram_111_PZD_12_12[3];
	HwOutputs.ST40_2_CMMT_2GF2_Promess_DO_SERVO_1_Siemens_telegram_111_PZD_12_12[4] := PlcOutputs.ST40_2_CMMT_2GF2_Promess_DO_SERVO_1_Siemens_telegram_111_PZD_12_12[4];
	HwOutputs.ST40_2_CMMT_2GF2_Promess_DO_SERVO_1_Siemens_telegram_111_PZD_12_12[5] := PlcOutputs.ST40_2_CMMT_2GF2_Promess_DO_SERVO_1_Siemens_telegram_111_PZD_12_12[5];
	HwOutputs.ST40_2_CMMT_2GF2_Promess_DO_SERVO_1_Siemens_telegram_111_PZD_12_12[6] := PlcOutputs.ST40_2_CMMT_2GF2_Promess_DO_SERVO_1_Siemens_telegram_111_PZD_12_12[6];
	HwOutputs.ST40_2_CMMT_2GF2_Promess_DO_SERVO_1_Siemens_telegram_111_PZD_12_12[7] := PlcOutputs.ST40_2_CMMT_2GF2_Promess_DO_SERVO_1_Siemens_telegram_111_PZD_12_12[7];
	HwOutputs.ST40_2_CMMT_2GF2_Promess_DO_SERVO_1_Siemens_telegram_111_PZD_12_12[8] := PlcOutputs.ST40_2_CMMT_2GF2_Promess_DO_SERVO_1_Siemens_telegram_111_PZD_12_12[8];
	HwOutputs.ST40_2_CMMT_2GF2_Promess_DO_SERVO_1_Siemens_telegram_111_PZD_12_12[9] := PlcOutputs.ST40_2_CMMT_2GF2_Promess_DO_SERVO_1_Siemens_telegram_111_PZD_12_12[9];
	HwOutputs.ST40_2_CMMT_2GF2_Promess_DO_SERVO_1_Siemens_telegram_111_PZD_12_12[10] := PlcOutputs.ST40_2_CMMT_2GF2_Promess_DO_SERVO_1_Siemens_telegram_111_PZD_12_12[10];
	HwOutputs.ST40_2_CMMT_2GF2_Promess_DO_SERVO_1_Siemens_telegram_111_PZD_12_12[11] := PlcOutputs.ST40_2_CMMT_2GF2_Promess_DO_SERVO_1_Siemens_telegram_111_PZD_12_12[11];
	HwOutputs.ST40_2_CMMT_2GF2_Promess_DO_SERVO_1_Siemens_telegram_111_PZD_12_12[12] := PlcOutputs.ST40_2_CMMT_2GF2_Promess_DO_SERVO_1_Siemens_telegram_111_PZD_12_12[12];
	HwOutputs.ST40_2_CMMT_2GF2_Promess_DO_SERVO_1_Siemens_telegram_111_PZD_12_12[13] := PlcOutputs.ST40_2_CMMT_2GF2_Promess_DO_SERVO_1_Siemens_telegram_111_PZD_12_12[13];
	HwOutputs.ST40_2_CMMT_2GF2_Promess_DO_SERVO_1_Siemens_telegram_111_PZD_12_12[14] := PlcOutputs.ST40_2_CMMT_2GF2_Promess_DO_SERVO_1_Siemens_telegram_111_PZD_12_12[14];
	HwOutputs.ST40_2_CMMT_2GF2_Promess_DO_SERVO_1_Siemens_telegram_111_PZD_12_12[15] := PlcOutputs.ST40_2_CMMT_2GF2_Promess_DO_SERVO_1_Siemens_telegram_111_PZD_12_12[15];
	HwOutputs.ST40_2_CMMT_2GF2_Promess_DO_SERVO_1_Siemens_telegram_111_PZD_12_12[16] := PlcOutputs.ST40_2_CMMT_2GF2_Promess_DO_SERVO_1_Siemens_telegram_111_PZD_12_12[16];
	HwOutputs.ST40_2_CMMT_2GF2_Promess_DO_SERVO_1_Siemens_telegram_111_PZD_12_12[17] := PlcOutputs.ST40_2_CMMT_2GF2_Promess_DO_SERVO_1_Siemens_telegram_111_PZD_12_12[17];
	HwOutputs.ST40_2_CMMT_2GF2_Promess_DO_SERVO_1_Siemens_telegram_111_PZD_12_12[18] := PlcOutputs.ST40_2_CMMT_2GF2_Promess_DO_SERVO_1_Siemens_telegram_111_PZD_12_12[18];
	HwOutputs.ST40_2_CMMT_2GF2_Promess_DO_SERVO_1_Siemens_telegram_111_PZD_12_12[19] := PlcOutputs.ST40_2_CMMT_2GF2_Promess_DO_SERVO_1_Siemens_telegram_111_PZD_12_12[19];
	HwOutputs.ST40_2_CMMT_2GF2_Promess_DO_SERVO_1_Siemens_telegram_111_PZD_12_12[20] := PlcOutputs.ST40_2_CMMT_2GF2_Promess_DO_SERVO_1_Siemens_telegram_111_PZD_12_12[20];
	HwOutputs.ST40_2_CMMT_2GF2_Promess_DO_SERVO_1_Siemens_telegram_111_PZD_12_12[21] := PlcOutputs.ST40_2_CMMT_2GF2_Promess_DO_SERVO_1_Siemens_telegram_111_PZD_12_12[21];
	HwOutputs.ST40_2_CMMT_2GF2_Promess_DO_SERVO_1_Siemens_telegram_111_PZD_12_12[22] := PlcOutputs.ST40_2_CMMT_2GF2_Promess_DO_SERVO_1_Siemens_telegram_111_PZD_12_12[22];
	HwOutputs.ST40_2_CMMT_2GF2_Promess_DO_SERVO_1_Siemens_telegram_111_PZD_12_12[23] := PlcOutputs.ST40_2_CMMT_2GF2_Promess_DO_SERVO_1_Siemens_telegram_111_PZD_12_12[23];
	HwOutputs.ST40_2_Promess_Menu_30_33_Out_1 := PlcOutputs.ST40_2_Promess_Menu_30_33_Out_1;
	HwOutputs.ST40_2_Promess_Menu_30_34_Out_1 := PlcOutputs.ST40_2_Promess_Menu_30_34_Out_1;
	HwOutputs.ST40_2_Promess_Menu_30_35_Out_1 := PlcOutputs.ST40_2_Promess_Menu_30_35_Out_1;
	HwOutputs.ST40_2_Promess_Menu_30_36_Out_1 := PlcOutputs.ST40_2_Promess_Menu_30_36_Out_1;
	HwOutputs.ST40_2_Promess_Menu_30_37_Out_1 := PlcOutputs.ST40_2_Promess_Menu_30_37_Out_1;
	HwOutputs.ST40_2_Promess_Menu_30_38_Out_1 := PlcOutputs.ST40_2_Promess_Menu_30_38_Out_1;
	HwOutputs.ST40_2_Promess_Menu_30_39_Out_1 := PlcOutputs.ST40_2_Promess_Menu_30_39_Out_1;
	HwOutputs.ST40_2_Promess_Menu_30_40_Out_1 := PlcOutputs.ST40_2_Promess_Menu_30_40_Out_1;
	HwOutputs.ST40_2_Promess_Menu_30_41_Out_1 := PlcOutputs.ST40_2_Promess_Menu_30_41_Out_1;
	HwOutputs.ST40_2_Promess_Menu_30_42_Out_1 := PlcOutputs.ST40_2_Promess_Menu_30_42_Out_1;
	HwOutputs.ST40_2_Promess_Menu_30_43_Out_1 := PlcOutputs.ST40_2_Promess_Menu_30_43_Out_1;
	HwOutputs.ST40_2_Promess_Menu_30_44_Out_1 := PlcOutputs.ST40_2_Promess_Menu_30_44_Out_1;
	HwOutputs.ST40_2_Promess_Menu_30_45_Out_1 := PlcOutputs.ST40_2_Promess_Menu_30_45_Out_1;
	HwOutputs.ST40_2_Promess_Menu_30_46_Out_1 := PlcOutputs.ST40_2_Promess_Menu_30_46_Out_1;
	HwOutputs.ST40_2_Promess_Menu_30_47_Out_1 := PlcOutputs.ST40_2_Promess_Menu_30_47_Out_1;
	HwOutputs.ST40_2_Promess_Menu_30_48_Out_1 := PlcOutputs.ST40_2_Promess_Menu_30_48_Out_1;
	HwOutputs.ST40_2_Promess_Menu_30_49_Out_1 := PlcOutputs.ST40_2_Promess_Menu_30_49_Out_1;
	HwOutputs.ST40_2_Promess_Menu_30_50_Out_1 := PlcOutputs.ST40_2_Promess_Menu_30_50_Out_1;
	HwOutputs.ST40_2_Promess_Menu_30_51_Out_1 := PlcOutputs.ST40_2_Promess_Menu_30_51_Out_1;
	HwOutputs.ST40_2_Promess_Menu_30_52_Out_1 := PlcOutputs.ST40_2_Promess_Menu_30_52_Out_1;
	HwOutputs.ST40_2_Promess_Menu_30_53_Out_1 := PlcOutputs.ST40_2_Promess_Menu_30_53_Out_1;
	HwOutputs.ST40_2_Promess_Menu_30_54_Out_1 := PlcOutputs.ST40_2_Promess_Menu_30_54_Out_1;
	HwOutputs.ST40_2_Promess_Menu_30_55_Out_1 := PlcOutputs.ST40_2_Promess_Menu_30_55_Out_1;
	HwOutputs.ST40_2_Promess_Menu_30_56_Out_1 := PlcOutputs.ST40_2_Promess_Menu_30_56_Out_1;
	HwOutputs.ST40_2_Promess_Menu_30_57_Out_1 := PlcOutputs.ST40_2_Promess_Menu_30_57_Out_1;
	HwOutputs.ST40_2_Promess_Menu_30_58_Out_1 := PlcOutputs.ST40_2_Promess_Menu_30_58_Out_1;
	HwOutputs.ST40_2_Promess_Menu_30_59_Out_1 := PlcOutputs.ST40_2_Promess_Menu_30_59_Out_1;
	HwOutputs.ST40_2_Promess_Menu_30_60_Out_1 := PlcOutputs.ST40_2_Promess_Menu_30_60_Out_1;
	HwOutputs.ST40_2_Promess_Menu_30_61_Out_1 := PlcOutputs.ST40_2_Promess_Menu_30_61_Out_1;
	HwOutputs.ST40_2_Promess_Menu_30_62_Out_1 := PlcOutputs.ST40_2_Promess_Menu_30_62_Out_1;
	HwOutputs.ST40_2_Promess_Menu_30_63_Out_1 := PlcOutputs.ST40_2_Promess_Menu_30_63_Out_1;
	HwOutputs.ST40_2_Promess_Menu_30_64_Out_1 := PlcOutputs.ST40_2_Promess_Menu_30_64_Out_1;
	HwOutputs.ST40_CPX_MPA1S_VMPA1_FB_EMS_8_8DO_1 := PlcOutputs.ST40_CPX_MPA1S_VMPA1_FB_EMS_8_8DO_1;
	HwOutputs.ST40_CPX_MPA1S_VMPA1_FB_EMS_8_8DO_2 := PlcOutputs.ST40_CPX_MPA1S_VMPA1_FB_EMS_8_8DO_2;
	HwOutputs.ST40_CPX_MPA1S_VMPA1_FB_EMS_8_8DO_3 := PlcOutputs.ST40_CPX_MPA1S_VMPA1_FB_EMS_8_8DO_3;
	HwOutputs.ST40_CPX_MPA1G_VMPA1_FB_EMG_8_8DO_1 := PlcOutputs.ST40_CPX_MPA1G_VMPA1_FB_EMG_8_8DO_1;
	HwOutputs.ST40_ET200SP_CM_4xIO_Link_1[0] := PlcOutputs.ST40_ET200SP_CM_4xIO_Link_1[0];
	HwOutputs.ST40_ET200SP_CM_4xIO_Link_1[1] := PlcOutputs.ST40_ET200SP_CM_4xIO_Link_1[1];
	HwOutputs.ST40_ET200SP_CM_4xIO_Link_1[2] := PlcOutputs.ST40_ET200SP_CM_4xIO_Link_1[2];
	HwOutputs.ST40_ET200SP_CM_4xIO_Link_1[3] := PlcOutputs.ST40_ET200SP_CM_4xIO_Link_1[3];
	HwOutputs.ST40_ET200SP_CM_4xIO_Link_1[4] := PlcOutputs.ST40_ET200SP_CM_4xIO_Link_1[4];
	HwOutputs.ST40_ET200SP_CM_4xIO_Link_1[5] := PlcOutputs.ST40_ET200SP_CM_4xIO_Link_1[5];
	HwOutputs.ST40_ET200SP_CM_4xIO_Link_1[6] := PlcOutputs.ST40_ET200SP_CM_4xIO_Link_1[6];
	HwOutputs.ST40_ET200SP_CM_4xIO_Link_1[7] := PlcOutputs.ST40_ET200SP_CM_4xIO_Link_1[7];
	HwOutputs.ST40_ET200SP_CM_4xIO_Link_1[8] := PlcOutputs.ST40_ET200SP_CM_4xIO_Link_1[8];
	HwOutputs.ST40_ET200SP_CM_4xIO_Link_1[9] := PlcOutputs.ST40_ET200SP_CM_4xIO_Link_1[9];
	HwOutputs.ST40_ET200SP_CM_4xIO_Link_1[10] := PlcOutputs.ST40_ET200SP_CM_4xIO_Link_1[10];
	HwOutputs.ST40_ET200SP_CM_4xIO_Link_1[11] := PlcOutputs.ST40_ET200SP_CM_4xIO_Link_1[11];
	HwOutputs.ST40_ET200SP_CM_4xIO_Link_1[12] := PlcOutputs.ST40_ET200SP_CM_4xIO_Link_1[12];
	HwOutputs.ST40_ET200SP_CM_4xIO_Link_1[13] := PlcOutputs.ST40_ET200SP_CM_4xIO_Link_1[13];
	HwOutputs.ST40_ET200SP_CM_4xIO_Link_1[14] := PlcOutputs.ST40_ET200SP_CM_4xIO_Link_1[14];
	HwOutputs.ST40_ET200SP_CM_4xIO_Link_1[15] := PlcOutputs.ST40_ET200SP_CM_4xIO_Link_1[15];
	HwOutputs.ST40_ET200SP_CM_4xIO_Link_1[16] := PlcOutputs.ST40_ET200SP_CM_4xIO_Link_1[16];
	HwOutputs.ST40_ET200SP_CM_4xIO_Link_1[17] := PlcOutputs.ST40_ET200SP_CM_4xIO_Link_1[17];
	HwOutputs.ST40_ET200SP_CM_4xIO_Link_1[18] := PlcOutputs.ST40_ET200SP_CM_4xIO_Link_1[18];
	HwOutputs.ST40_ET200SP_CM_4xIO_Link_1[19] := PlcOutputs.ST40_ET200SP_CM_4xIO_Link_1[19];
	HwOutputs.ST40_ET200SP_CM_4xIO_Link_1[20] := PlcOutputs.ST40_ET200SP_CM_4xIO_Link_1[20];
	HwOutputs.ST40_ET200SP_CM_4xIO_Link_1[21] := PlcOutputs.ST40_ET200SP_CM_4xIO_Link_1[21];
	HwOutputs.ST40_ET200SP_CM_4xIO_Link_1[22] := PlcOutputs.ST40_ET200SP_CM_4xIO_Link_1[22];
	HwOutputs.ST40_ET200SP_CM_4xIO_Link_1[23] := PlcOutputs.ST40_ET200SP_CM_4xIO_Link_1[23];
	HwOutputs.ST40_ET200SP_CM_4xIO_Link_1[24] := PlcOutputs.ST40_ET200SP_CM_4xIO_Link_1[24];
	HwOutputs.ST40_ET200SP_CM_4xIO_Link_1[25] := PlcOutputs.ST40_ET200SP_CM_4xIO_Link_1[25];
	HwOutputs.ST40_ET200SP_CM_4xIO_Link_1[26] := PlcOutputs.ST40_ET200SP_CM_4xIO_Link_1[26];
	HwOutputs.ST40_ET200SP_CM_4xIO_Link_1[27] := PlcOutputs.ST40_ET200SP_CM_4xIO_Link_1[27];
	HwOutputs.ST40_ET200SP_CM_4xIO_Link_1[28] := PlcOutputs.ST40_ET200SP_CM_4xIO_Link_1[28];
	HwOutputs.ST40_ET200SP_CM_4xIO_Link_1[29] := PlcOutputs.ST40_ET200SP_CM_4xIO_Link_1[29];
	HwOutputs.ST40_ET200SP_CM_4xIO_Link_1[30] := PlcOutputs.ST40_ET200SP_CM_4xIO_Link_1[30];
	HwOutputs.ST40_ET200SP_CM_4xIO_Link_1[31] := PlcOutputs.ST40_ET200SP_CM_4xIO_Link_1[31];
	HwOutputs.ST40_ET200SP_CM_4xIO_Link_2[0] := PlcOutputs.ST40_ET200SP_CM_4xIO_Link_2[0];
	HwOutputs.ST40_ET200SP_CM_4xIO_Link_2[1] := PlcOutputs.ST40_ET200SP_CM_4xIO_Link_2[1];
	HwOutputs.ST40_ET200SP_CM_4xIO_Link_2[2] := PlcOutputs.ST40_ET200SP_CM_4xIO_Link_2[2];
	HwOutputs.ST40_ET200SP_CM_4xIO_Link_2[3] := PlcOutputs.ST40_ET200SP_CM_4xIO_Link_2[3];
	HwOutputs.ST40_ET200SP_CM_4xIO_Link_2[4] := PlcOutputs.ST40_ET200SP_CM_4xIO_Link_2[4];
	HwOutputs.ST40_ET200SP_CM_4xIO_Link_2[5] := PlcOutputs.ST40_ET200SP_CM_4xIO_Link_2[5];
	HwOutputs.ST40_ET200SP_CM_4xIO_Link_2[6] := PlcOutputs.ST40_ET200SP_CM_4xIO_Link_2[6];
	HwOutputs.ST40_ET200SP_CM_4xIO_Link_2[7] := PlcOutputs.ST40_ET200SP_CM_4xIO_Link_2[7];
	HwOutputs.ST40_ET200SP_CM_4xIO_Link_2[8] := PlcOutputs.ST40_ET200SP_CM_4xIO_Link_2[8];
	HwOutputs.ST40_ET200SP_CM_4xIO_Link_2[9] := PlcOutputs.ST40_ET200SP_CM_4xIO_Link_2[9];
	HwOutputs.ST40_ET200SP_CM_4xIO_Link_2[10] := PlcOutputs.ST40_ET200SP_CM_4xIO_Link_2[10];
	HwOutputs.ST40_ET200SP_CM_4xIO_Link_2[11] := PlcOutputs.ST40_ET200SP_CM_4xIO_Link_2[11];
	HwOutputs.ST40_ET200SP_CM_4xIO_Link_2[12] := PlcOutputs.ST40_ET200SP_CM_4xIO_Link_2[12];
	HwOutputs.ST40_ET200SP_CM_4xIO_Link_2[13] := PlcOutputs.ST40_ET200SP_CM_4xIO_Link_2[13];
	HwOutputs.ST40_ET200SP_CM_4xIO_Link_2[14] := PlcOutputs.ST40_ET200SP_CM_4xIO_Link_2[14];
	HwOutputs.ST40_ET200SP_CM_4xIO_Link_2[15] := PlcOutputs.ST40_ET200SP_CM_4xIO_Link_2[15];
	HwOutputs.ST40_ET200SP_CM_4xIO_Link_2[16] := PlcOutputs.ST40_ET200SP_CM_4xIO_Link_2[16];
	HwOutputs.ST40_ET200SP_CM_4xIO_Link_2[17] := PlcOutputs.ST40_ET200SP_CM_4xIO_Link_2[17];
	HwOutputs.ST40_ET200SP_CM_4xIO_Link_2[18] := PlcOutputs.ST40_ET200SP_CM_4xIO_Link_2[18];
	HwOutputs.ST40_ET200SP_CM_4xIO_Link_2[19] := PlcOutputs.ST40_ET200SP_CM_4xIO_Link_2[19];
	HwOutputs.ST40_ET200SP_CM_4xIO_Link_2[20] := PlcOutputs.ST40_ET200SP_CM_4xIO_Link_2[20];
	HwOutputs.ST40_ET200SP_CM_4xIO_Link_2[21] := PlcOutputs.ST40_ET200SP_CM_4xIO_Link_2[21];
	HwOutputs.ST40_ET200SP_CM_4xIO_Link_2[22] := PlcOutputs.ST40_ET200SP_CM_4xIO_Link_2[22];
	HwOutputs.ST40_ET200SP_CM_4xIO_Link_2[23] := PlcOutputs.ST40_ET200SP_CM_4xIO_Link_2[23];
	HwOutputs.ST40_ET200SP_CM_4xIO_Link_2[24] := PlcOutputs.ST40_ET200SP_CM_4xIO_Link_2[24];
	HwOutputs.ST40_ET200SP_CM_4xIO_Link_2[25] := PlcOutputs.ST40_ET200SP_CM_4xIO_Link_2[25];
	HwOutputs.ST40_ET200SP_CM_4xIO_Link_2[26] := PlcOutputs.ST40_ET200SP_CM_4xIO_Link_2[26];
	HwOutputs.ST40_ET200SP_CM_4xIO_Link_2[27] := PlcOutputs.ST40_ET200SP_CM_4xIO_Link_2[27];
	HwOutputs.ST40_ET200SP_CM_4xIO_Link_2[28] := PlcOutputs.ST40_ET200SP_CM_4xIO_Link_2[28];
	HwOutputs.ST40_ET200SP_CM_4xIO_Link_2[29] := PlcOutputs.ST40_ET200SP_CM_4xIO_Link_2[29];
	HwOutputs.ST40_ET200SP_CM_4xIO_Link_2[30] := PlcOutputs.ST40_ET200SP_CM_4xIO_Link_2[30];
	HwOutputs.ST40_ET200SP_CM_4xIO_Link_2[31] := PlcOutputs.ST40_ET200SP_CM_4xIO_Link_2[31];
	HwOutputs.ST40_ET200SP_DQ_16x24VDC_0_5A_ST_1 := PlcOutputs.ST40_ET200SP_DQ_16x24VDC_0_5A_ST_1;
	HwOutputs.ST40_ET200SP_DQ_8x24VDC_0_5A_ST_2 := PlcOutputs.ST40_ET200SP_DQ_8x24VDC_0_5A_ST_2;
	HwOutputs.ST40_ET200SP_DQ_8x24VDC_0_5A_ST_3 := PlcOutputs.ST40_ET200SP_DQ_8x24VDC_0_5A_ST_3;
END_FUNCTION
